// TIA Portal V15.1 export
// export: Created 2024-06-21T08:41:00.3129573Z, ExportSetting WithDefaults, DisplayName Totally Integrated Automation Portal, DisplayVersion V15.1 Update 5, DisplayName TIA Portal Openness, DisplayVersion V15.1 Update 5, DisplayName SINAMICS Startdrive Advanced, DisplayVersion V15.1, DisplayName G130, G150, S120, S150, SINAMICS MV, S210, DisplayVersion V15.1, DisplayName G110M, G120, G120C, G120D, G120P, DisplayVersion V15.1, DisplayName STEP 7 Professional, DisplayVersion V15.1 Update 5, DisplayName STEP 7 Safety, DisplayVersion V15.1, DisplayName WinCC Professional, DisplayVersion V15.1 Update 5, DisplayName SIMATIC Visualization Architect, DisplayVersion V15.1
FUNCTION_BLOCK "LVDComMasterS7-1500"   // FB2210, FBD
TITLE = LVDComMasterPNS7-1500
{ S7_Optimized_Access := 'FALSE' }
AUTHOR : VCC
FAMILY : Communic
VERSION : 0.1
// =============================================================================
// This module Is Used To Read & Send Data With VDCom Protocol
// =============================================================================
// stored: AutoNumber false, IsIECCheckEnabled false, SetENOAutomatically False, UDAEnableTagReadback false
   VAR_INPUT
      I_VDCommRecvDB { ExternalAccessible := 'False'; ExternalVisible := 'False'; ExternalWritable := 'False'} : DB_ANY;   // VD Communication Master DB
      I_VDCommSendDB { ExternalAccessible := 'False'; ExternalVisible := 'False'; ExternalWritable := 'False'} : DB_ANY;   // VD Communication Master DB
   END_VAR
   VAR_OUTPUT
      O_AlarmA { ExternalAccessible := 'False'; ExternalVisible := 'False'; ExternalWritable := 'False'} : Bool;   // Alarm A
      O_AlarmB { ExternalAccessible := 'False'; ExternalVisible := 'False'; ExternalWritable := 'False'} : Bool;   // Alarm B
      O_AlarmC { ExternalAccessible := 'False'; ExternalVisible := 'False'; ExternalWritable := 'False'} : Bool;   // Alarm C
      O_AlarmD { ExternalAccessible := 'False'; ExternalVisible := 'False'; ExternalWritable := 'False'} : Bool;   // Alarm D
      H_AlarmWord { ExternalAccessible := 'False'; ExternalVisible := 'False'; ExternalWritable := 'False'} : DWord;   // HMI Animation
   END_VAR
   VAR_IN_OUT
      IO_Alarm : "Alarm";   // Alarm
      IO_VD : "VDComm";
      IO_ConnectionSetting : Variant;   // Software Connection Settings
      "H_VDComMasterPNS7-1500" : "H_VDComMasterPNS7-1500";   // Animation
   END_VAR
   VAR DB_SPECIFIC
      AD_SendTimeOut { ExternalAccessible := 'False'; ExternalVisible := 'False'; ExternalWritable := 'False'} : Bool;   // Communication Error Send Condition Active Too Long / Kommunikationsfel Sändvillkor Aktivt För Länge
      AD_VersionError { ExternalAccessible := 'False'; ExternalVisible := 'False'; ExternalWritable := 'False'} : Bool;   // Wrong Version Number / Fel Versionsnummer
      AD_ConnError { ExternalAccessible := 'False'; ExternalVisible := 'False'; ExternalWritable := 'False'} : Bool;   // Communication Error Connecting Or Disconnecting / Kommunikationsfel Uppkoppling Eller Nerkoppling
      AD_TCONConnected { ExternalAccessible := 'False'; ExternalVisible := 'False'; ExternalWritable := 'False'} : Bool;   // Not Connected / Ej Uppkopplad
      AD_TSENDError { ExternalAccessible := 'False'; ExternalVisible := 'False'; ExternalWritable := 'False'} : Bool;   // Error Transmission / Fel Sändning
      AD_TRECVError { ExternalAccessible := 'False'; ExternalVisible := 'False'; ExternalWritable := 'False'} : Bool;   // Error Receiving / Fel Mottagning
      AD_NoAckReceived { ExternalAccessible := 'False'; ExternalVisible := 'False'; ExternalWritable := 'False'} : Bool;   // Error On Ack Message / Fel Vid Ack Meddelande
      AD_SequenceNumberNok { ExternalAccessible := 'False'; ExternalVisible := 'False'; ExternalWritable := 'False'} : Bool;   // Incorrect Sequence Number / Felaktigt Sekvensnummer
      AD_TimeoutApplMsgMem { ExternalAccessible := 'False'; ExternalVisible := 'False'; ExternalWritable := 'False'} : Bool;   // Timeout Message To Subsystem / Timeout Meddelande Till Subsystem
      HMIManual { ExternalAccessible := 'False'; ExternalVisible := 'False'; ExternalWritable := 'False'} : Bool;   // Connect or disconnect manual via HMI
      HMIResetAndInit { ExternalAccessible := 'False'; ExternalVisible := 'False'; ExternalWritable := 'False'} : Bool;   // Reset Alarms from HMI
      HMIConnect { ExternalAccessible := 'False'; ExternalVisible := 'False'; ExternalWritable := 'False'} : Bool;   // Connect from HMI
      HMIDisConnect { ExternalAccessible := 'False'; ExternalVisible := 'False'; ExternalWritable := 'False'} : Bool;   // DisConnect from HMI
      Manual { ExternalAccessible := 'False'; ExternalVisible := 'False'; ExternalWritable := 'False'} : Bool;   // Connect or disconnect manual via HMI
      SendActive { ExternalAccessible := 'False'; ExternalVisible := 'False'; ExternalWritable := 'False'} : Bool;   // Sending is Active
      NdrDelayed { ExternalAccessible := 'False'; ExternalVisible := 'False'; ExternalWritable := 'False'} : Bool;   // Time required to elapse before to send acknowledge
      KeepAliveReq { ExternalAccessible := 'False'; ExternalVisible := 'False'; ExternalWritable := 'False'} : Bool;   // Request to send keep alive message
      AckRcvd { ExternalAccessible := 'False'; ExternalVisible := 'False'; ExternalWritable := 'False'} : Bool;   // Acknowledge Received
      SeqNbrOk { ExternalAccessible := 'False'; ExternalVisible := 'False'; ExternalWritable := 'False'} : Bool;   // Sequence number in received message is the same as sended
      AckOk { ExternalAccessible := 'False'; ExternalVisible := 'False'; ExternalWritable := 'False'} : Bool;   // Received acknowledge message ok
      AckNok { ExternalAccessible := 'False'; ExternalVisible := 'False'; ExternalWritable := 'False'} : Bool;   // Received acknowledge message not ok
      NewMessage { ExternalAccessible := 'False'; ExternalVisible := 'False'; ExternalWritable := 'False'} : Bool;   // New Data Message has been received
      SendInactive { ExternalAccessible := 'False'; ExternalVisible := 'False'; ExternalWritable := 'False'} : Bool;   // Sending inActive
      SendJobCompleted { ExternalAccessible := 'False'; ExternalVisible := 'False'; ExternalWritable := 'False'} : Bool;   // Status of the TSEND module: Job Completed no job active
      SendStartOfProc { ExternalAccessible := 'False'; ExternalVisible := 'False'; ExternalWritable := 'False'} : Bool;   // Status of TSEND: Start of Processing
      SendFollowOnCall { ExternalAccessible := 'False'; ExternalVisible := 'False'; ExternalWritable := 'False'} : Bool;   // Status of TSEND: Followon calls being processed
      SendNackMem { ExternalAccessible := 'False'; ExternalVisible := 'False'; ExternalWritable := 'False'} : Bool;   // Command to send Not acknowledge message
      SendNackPulse { ExternalAccessible := 'False'; ExternalVisible := 'False'; ExternalWritable := 'False'} : Bool;   // Pulse to send the Not Acknowledge message
      SendNackCmd { ExternalAccessible := 'False'; ExternalVisible := 'False'; ExternalWritable := 'False'} : Bool;   // Command to send a NOT Acknowledge message
      SendAckMem { ExternalAccessible := 'False'; ExternalVisible := 'False'; ExternalWritable := 'False'} : Bool;   // Command to send Acknowledge message
      SendAckPulse { ExternalAccessible := 'False'; ExternalVisible := 'False'; ExternalWritable := 'False'} : Bool;   // Pulse to send Acknowledge message
      SendAckCmd { ExternalAccessible := 'False'; ExternalVisible := 'False'; ExternalWritable := 'False'} : Bool;   // Command to send an Acknowledge message
      SendKeepAliveMem { ExternalAccessible := 'False'; ExternalVisible := 'False'; ExternalWritable := 'False'} : Bool;   // Command to send the keep alive signal
      SendKeepAlivePulse { ExternalAccessible := 'False'; ExternalVisible := 'False'; ExternalWritable := 'False'} : Bool;   // Pulse to send keep alive message
      SendKeepAliveCmd { ExternalAccessible := 'False'; ExternalVisible := 'False'; ExternalWritable := 'False'} : Bool;   // Command to Send Keep Alive message
      SendApplMsgMem { ExternalAccessible := 'False'; ExternalVisible := 'False'; ExternalWritable := 'False'} : Bool;   // Command to send apllication data
      SendApplMsgPulse { ExternalAccessible := 'False'; ExternalVisible := 'False'; ExternalWritable := 'False'} : Bool;   // Pulse created upon SendApplMsgCmd
      SendApplMsgCmd { ExternalAccessible := 'False'; ExternalVisible := 'False'; ExternalWritable := 'False'} : Bool;   // Command to send an Application message
      NewMsgNbr { ExternalAccessible := 'False'; ExternalVisible := 'False'; ExternalWritable := 'False'} : Bool;   // Message number of last received message
      NackIsLastSent { ExternalAccessible := 'False'; ExternalVisible := 'False'; ExternalWritable := 'False'} : Bool;   // Memorise that Nack was send
      DupplMsg { ExternalAccessible := 'False'; ExternalVisible := 'False'; ExternalWritable := 'False'} : Bool;   // When received msg number is the same as previous
      RecvLenOK { ExternalAccessible := 'False'; ExternalVisible := 'False'; ExternalWritable := 'False'} : Bool;   // If protocol Len and actual received msg are the same
      WaitForAck { ExternalAccessible := 'False'; ExternalVisible := 'False'; ExternalWritable := 'False'} : Bool;   // State waiting for acknowledge
      TimeOutTConn { ExternalAccessible := 'False'; ExternalVisible := 'False'; ExternalWritable := 'False'} : Bool;   // Time out on connecting or disconnecting
      TimeoutTCON { ExternalAccessible := 'False'; ExternalVisible := 'False'; ExternalWritable := 'False'} : Bool;   // Memory of connection time out
      TimeoutTDISCON { ExternalAccessible := 'False'; ExternalVisible := 'False'; ExternalWritable := 'False'} : Bool;   // Time out on disconnecting
      TimeoutApplMsg { ExternalAccessible := 'False'; ExternalVisible := 'False'; ExternalWritable := 'False'} : Bool;   // Time Out on apllication message, no ack received
      DisconnConn { ExternalAccessible := 'False'; ExternalVisible := 'False'; ExternalWritable := 'False'} : Bool;   // Time before connecting after disconnecting
      Edge { ExternalAccessible := 'False'; ExternalVisible := 'False'; ExternalWritable := 'False'} : Bool;   // Positive edge Detection for connected
      ResetAppliMsgCnt { ExternalAccessible := 'False'; ExternalVisible := 'False'; ExternalWritable := 'False'} : Bool;   // Reset the Application message counter
      ResetKeepAliveCnt { ExternalAccessible := 'False'; ExternalVisible := 'False'; ExternalWritable := 'False'} : Bool;   // Reset the keep alive counter
      ResetAckCmdCnt { ExternalAccessible := 'False'; ExternalVisible := 'False'; ExternalWritable := 'False'} : Bool;   // Reset the acknowledge counter
      ResetNackCmdCnt { ExternalAccessible := 'False'; ExternalVisible := 'False'; ExternalWritable := 'False'} : Bool;   // Reset the Nacknowledge counter
      ResetAckRcvCnt { ExternalAccessible := 'False'; ExternalVisible := 'False'; ExternalWritable := 'False'} : Bool;   // Reset the received Ack counter
      ResetDataMsgCnt { ExternalAccessible := 'False'; ExternalVisible := 'False'; ExternalWritable := 'False'} : Bool;   // Reset the received Data message counter
      ResetSeqNokCnt { ExternalAccessible := 'False'; ExternalVisible := 'False'; ExternalWritable := 'False'} : Bool;   // Reset the sequence nok counter
      ResetSendActive { ExternalAccessible := 'False'; ExternalVisible := 'False'; ExternalWritable := 'False'} : Bool;   // Reset Send Active due to time out
      SendDone { ExternalAccessible := 'False'; ExternalVisible := 'False'; ExternalWritable := 'False'} : Bool;   // Reset the Ndr counter on overrun
      DelayOpen { ExternalAccessible := 'False'; ExternalVisible := 'False'; ExternalWritable := 'False'} : Bool;   // Delay Start Connect
      DelayConn { ExternalAccessible := 'False'; ExternalVisible := 'False'; ExternalWritable := 'False'} : Bool;   // Delay Connected
      AlarmA { ExternalAccessible := 'False'; ExternalVisible := 'False'; ExternalWritable := 'False'} : Bool;   // Alarm A
      AlarmB { ExternalAccessible := 'False'; ExternalVisible := 'False'; ExternalWritable := 'False'} : Bool;   // Alarm B
      AlarmC { ExternalAccessible := 'False'; ExternalVisible := 'False'; ExternalWritable := 'False'} : Bool;   // Alarm C
      AlarmD { ExternalAccessible := 'False'; ExternalVisible := 'False'; ExternalWritable := 'False'} : Bool;   // Alarm D
      OldSubSystem { ExternalAccessible := 'False'; ExternalVisible := 'False'; ExternalWritable := 'False'} : Word;   // Memorise last received subsystem address
      OldRecMsgNbr { ExternalAccessible := 'False'; ExternalVisible := 'False'; ExternalWritable := 'False'} : Word := W#16#999;   // Memorise the last message number
      SendMsgNbr { ExternalAccessible := 'False'; ExternalVisible := 'False'; ExternalWritable := 'False'} : Word;   // Number is incremented for each msg and Reset to 1 when > 1000
      RecvLen { ExternalAccessible := 'False'; ExternalVisible := 'False'; ExternalWritable := 'False'} : Int;   // Memory of the received data length
      RecvDBNbr { ExternalAccessible := 'False'; ExternalVisible := 'False'; ExternalWritable := 'False'} : Int;   // Receive DB Number
      SendDBNbr { ExternalAccessible := 'False'; ExternalVisible := 'False'; ExternalWritable := 'False'} : Int;   // Send DB Number
      SendApplMsgCnt { ExternalAccessible := 'False'; ExternalVisible := 'False'; ExternalWritable := 'False'} : Int;   // Counting number of Application messages
      SendKeepAliveCnt { ExternalAccessible := 'False'; ExternalVisible := 'False'; ExternalWritable := 'False'} : Int;   // Counting number of keep alive messages
      SendAckCmdCnt { ExternalAccessible := 'False'; ExternalVisible := 'False'; ExternalWritable := 'False'} : Int;   // Counting the number of Ack messages
      SendNackCmdCnt { ExternalAccessible := 'False'; ExternalVisible := 'False'; ExternalWritable := 'False'} : Int;   // Counting the number of Nack messages
      RcvAckCnt { ExternalAccessible := 'False'; ExternalVisible := 'False'; ExternalWritable := 'False'} : Int;   // Counting the number of received Ack messages
      RcvDataMsgCnt { ExternalAccessible := 'False'; ExternalVisible := 'False'; ExternalWritable := 'False'} : Int;   // Counting the number of Data messages
      SeqNokCnt { ExternalAccessible := 'False'; ExternalVisible := 'False'; ExternalWritable := 'False'} : Int;   // Counter indicating the number of received sequence errors
      NdrCnt { ExternalAccessible := 'False'; ExternalVisible := 'False'; ExternalWritable := 'False'} : Int;   // Counter indicating the all received events
   END_VAR
   VAR
      TConVD { ExternalAccessible := 'False'; ExternalVisible := 'False'; ExternalWritable := 'False'; S7_SetPoint := 'True'} : TCON;   // Connect
      TDisConVD { ExternalAccessible := 'False'; ExternalVisible := 'False'; ExternalWritable := 'False'; S7_SetPoint := 'True'} : TDISCON;   // Disconnect
      TRcvVDData { ExternalAccessible := 'False'; ExternalVisible := 'False'; ExternalWritable := 'False'; S7_SetPoint := 'True'} : TRCV;   // Receive
      TSendVD { ExternalAccessible := 'False'; ExternalVisible := 'False'; ExternalWritable := 'False'; S7_SetPoint := 'True'} : TSEND;   // Send
   END_VAR
   VAR DB_SPECIFIC
      TCON { ExternalAccessible := 'False'; ExternalVisible := 'False'; ExternalWritable := 'False'} : Struct   // Structure
         Connecting { ExternalAccessible := 'False'; ExternalVisible := 'False'; ExternalWritable := 'False'} : Bool;
         Connected { ExternalAccessible := 'False'; ExternalVisible := 'False'; ExternalWritable := 'False'} : Bool;
         Done { ExternalAccessible := 'False'; ExternalVisible := 'False'; ExternalWritable := 'False'} : Bool;
         Busy { ExternalAccessible := 'False'; ExternalVisible := 'False'; ExternalWritable := 'False'} : Bool;
         Error { ExternalAccessible := 'False'; ExternalVisible := 'False'; ExternalWritable := 'False'} : Bool;
         Req { ExternalAccessible := 'False'; ExternalVisible := 'False'; ExternalWritable := 'False'} : Bool;
         Status { ExternalAccessible := 'False'; ExternalVisible := 'False'; ExternalWritable := 'False'} : Word;
         Status_Mem { ExternalAccessible := 'False'; ExternalVisible := 'False'; ExternalWritable := 'False'} : Word;
         Status_Int { ExternalAccessible := 'False'; ExternalVisible := 'False'; ExternalWritable := 'False'} : Int;
      END_STRUCT;
      TDISCON { ExternalAccessible := 'False'; ExternalVisible := 'False'; ExternalWritable := 'False'} : Struct   // Structure
         Disconnecting { ExternalAccessible := 'False'; ExternalVisible := 'False'; ExternalWritable := 'False'} : Bool;
         Done { ExternalAccessible := 'False'; ExternalVisible := 'False'; ExternalWritable := 'False'} : Bool;
         Busy { ExternalAccessible := 'False'; ExternalVisible := 'False'; ExternalWritable := 'False'} : Bool;
         Error { ExternalAccessible := 'False'; ExternalVisible := 'False'; ExternalWritable := 'False'} : Bool;
         Req { ExternalAccessible := 'False'; ExternalVisible := 'False'; ExternalWritable := 'False'} : Bool;
         Status { ExternalAccessible := 'False'; ExternalVisible := 'False'; ExternalWritable := 'False'} : Word;
         Status_Mem { ExternalAccessible := 'False'; ExternalVisible := 'False'; ExternalWritable := 'False'} : Word;
      END_STRUCT;
      TRECV { ExternalAccessible := 'False'; ExternalVisible := 'False'; ExternalWritable := 'False'} : Struct   // Structure
         Receiving { ExternalAccessible := 'False'; ExternalVisible := 'False'; ExternalWritable := 'False'} : Bool;
         Ndr { ExternalAccessible := 'False'; ExternalVisible := 'False'; ExternalWritable := 'False'} : Bool;
         Busy { ExternalAccessible := 'False'; ExternalVisible := 'False'; ExternalWritable := 'False'} : Bool;
         Error { ExternalAccessible := 'False'; ExternalVisible := 'False'; ExternalWritable := 'False'} : Bool;
         RcvConError { ExternalAccessible := 'False'; ExternalVisible := 'False'; ExternalWritable := 'False'} : Bool;
         Status { ExternalAccessible := 'False'; ExternalVisible := 'False'; ExternalWritable := 'False'} : Word;
         Status_Mem { ExternalAccessible := 'False'; ExternalVisible := 'False'; ExternalWritable := 'False'} : Word;
         Length { ExternalAccessible := 'False'; ExternalVisible := 'False'; ExternalWritable := 'False'} : UDInt;
      END_STRUCT;
      TSEND { ExternalAccessible := 'False'; ExternalVisible := 'False'; ExternalWritable := 'False'} : Struct   // Structure
         Sending { ExternalAccessible := 'False'; ExternalVisible := 'False'; ExternalWritable := 'False'} : Bool;
         Done { ExternalAccessible := 'False'; ExternalVisible := 'False'; ExternalWritable := 'False'} : Bool;
         Busy { ExternalAccessible := 'False'; ExternalVisible := 'False'; ExternalWritable := 'False'} : Bool;
         Error { ExternalAccessible := 'False'; ExternalVisible := 'False'; ExternalWritable := 'False'} : Bool;
         Status { ExternalAccessible := 'False'; ExternalVisible := 'False'; ExternalWritable := 'False'} : Word;
         Status_Mem { ExternalAccessible := 'False'; ExternalVisible := 'False'; ExternalWritable := 'False'} : Word;
      END_STRUCT;
      NackCmdCntr { ExternalAccessible := 'False'; ExternalVisible := 'False'; ExternalWritable := 'False'; S7_SetPoint := 'True'} : CTU_INT;   // Count number of NotAck messages send by PLC
      AckCmdCnt { ExternalAccessible := 'False'; ExternalVisible := 'False'; ExternalWritable := 'False'; S7_SetPoint := 'True'} : CTU_INT;   // Count number of Ack messages send by PLC
      KeepAliveCnt { ExternalAccessible := 'False'; ExternalVisible := 'False'; ExternalWritable := 'False'; S7_SetPoint := 'True'} : CTU_INT;   // Count number of Keep Alived Messages send by PLC
      AppliMsgCnt { ExternalAccessible := 'False'; ExternalVisible := 'False'; ExternalWritable := 'False'; S7_SetPoint := 'True'} : CTU_INT;   // Count number of Application messages send by PLC
      AckRvcCntr { ExternalAccessible := 'False'; ExternalVisible := 'False'; ExternalWritable := 'False'; S7_SetPoint := 'True'} : CTU_INT;   // Count number of Ack messages received
      DataMsgRcvCntr { ExternalAccessible := 'False'; ExternalVisible := 'False'; ExternalWritable := 'False'; S7_SetPoint := 'True'} : CTU_INT;   // Count number of data messages received
      SeqNumNok { ExternalAccessible := 'False'; ExternalVisible := 'False'; ExternalWritable := 'False'; S7_SetPoint := 'True'} : CTU_INT;   // counter to know the sequence number errors
      NdrPace { ExternalAccessible := 'False'; ExternalVisible := 'False'; ExternalWritable := 'False'; S7_SetPoint := 'True'} : TOF_TIME;   // Make sure that not too many messages are received at once
      TimeOutSending { ExternalAccessible := 'False'; ExternalVisible := 'False'; ExternalWritable := 'False'; S7_SetPoint := 'True'} : TON_TIME;   // TimeOut on Send operation
      TimeOutAckApplMsg { ExternalAccessible := 'False'; ExternalVisible := 'False'; ExternalWritable := 'False'; S7_SetPoint := 'True'} : TON_TIME;   // Timeout on reception of Ack on Application message
      TimeOutOnConnection { ExternalAccessible := 'False'; ExternalVisible := 'False'; ExternalWritable := 'False'; S7_SetPoint := 'True'} : TON_TIME;   // TimeOut on connecting
      KeepAliveFreq { ExternalAccessible := 'False'; ExternalVisible := 'False'; ExternalWritable := 'False'; S7_SetPoint := 'True'} : TON_TIME;   // Timer to timeout the keep alive messages
      DisconnectRequest { ExternalAccessible := 'False'; ExternalVisible := 'False'; ExternalWritable := 'False'; S7_SetPoint := 'True'} : TON_TIME;   // Request to disconnect after timeout
      WaitingForAck { ExternalAccessible := 'False'; ExternalVisible := 'False'; ExternalWritable := 'False'; S7_SetPoint := 'True'} : TON_TIME;   // Waiting for Ack to receive
      SubSystResponseTimeOut { ExternalAccessible := 'False'; ExternalVisible := 'False'; ExternalWritable := 'False'; S7_SetPoint := 'True'} : TON_TIME;   // TimeOut subsystem reply
      TimeOutSendActive { ExternalAccessible := 'False'; ExternalVisible := 'False'; ExternalWritable := 'False'; S7_SetPoint := 'True'} : TON_TIME;   // When SendActive is ON for too long
      DelayStartConnect { ExternalAccessible := 'False'; ExternalVisible := 'False'; ExternalWritable := 'False'; S7_SetPoint := 'True'} : TON_TIME;   // FB
      DelayConnected { ExternalAccessible := 'False'; ExternalVisible := 'False'; ExternalWritable := 'False'; S7_SetPoint := 'True'} : TON_TIME;   // FB
   END_VAR
   VAR
      _VDConManual { ExternalAccessible := 'False'; ExternalVisible := 'False'; ExternalWritable := 'False'; S7_SetPoint := 'True'} : "LToggle";   // FB
   END_VAR
   VAR DB_SPECIFIC
      ConnectionSettings { ExternalAccessible := 'False'; ExternalVisible := 'False'; ExternalWritable := 'False'; S7_SetPoint := 'True'} : TCON_Param;   // Structrure
   END_VAR
   VAR_TEMP
      PointerRecv : Any;   // Pointer to receive buffer
      PointerSend : Any;   // Pointer to Send Buffer
      PointerSendBuf : Any;   // Pointer to Send buffer
      OutBuf : Int;   // Integer to select the Send buffer
      UserMsgType : Bool;   // Message Type
      RecvTimeOut : Bool;   // Receive Time Out
      MsgLen : UDInt;   // Message length
      MessageLengthRecv : Int;   // Message Length receive
      TempIntStatus : Int;   // for type casting to integer
      TempInt : Int;   // for type casting to integer
      RecvDBNO : UInt;
      LengthDB : UDInt;
      TempBool : Array[1..16] of Bool;
      ConnectionSetting : Variant;
   END_VAR
   VAR_TEMP   // added for the SCL form of the ladder/FBD networks
      _w1 : Bool;
      _w2 : Bool;
   END_VAR
BEGIN

REGION Network 1: **** 1 - Inputs **** Extract the selection from HMI
   // Extract the selection from HMI
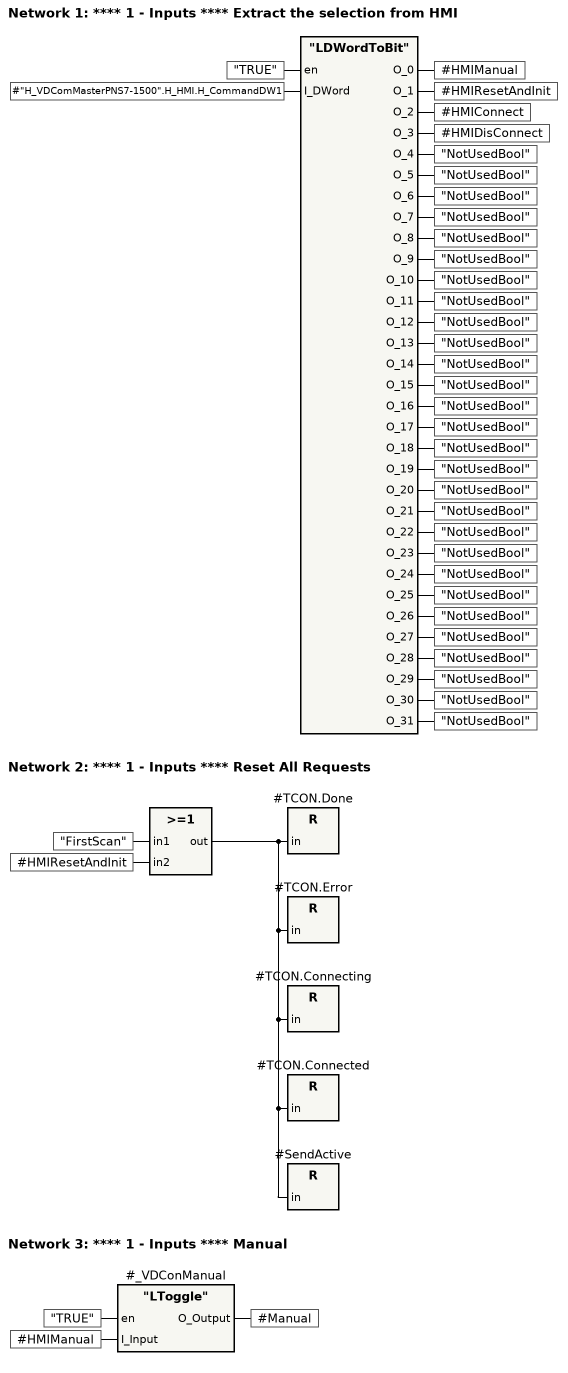
   IF "TRUE" THEN
       "LDWordToBit"(I_DWord := #"H_VDComMasterPNS7-1500".H_HMI.H_CommandDW1,
                     O_0 => #HMIManual,
                     O_1 => #HMIResetAndInit,
                     O_2 => #HMIConnect,
                     O_3 => #HMIDisConnect,
                     O_4 => "NotUsedBool",
                     O_5 => "NotUsedBool",
                     O_6 => "NotUsedBool",
                     O_7 => "NotUsedBool",
                     O_8 => "NotUsedBool",
                     O_9 => "NotUsedBool",
                     O_10 => "NotUsedBool",
                     O_11 => "NotUsedBool",
                     O_12 => "NotUsedBool",
                     O_13 => "NotUsedBool",
                     O_14 => "NotUsedBool",
                     O_15 => "NotUsedBool",
                     O_16 => "NotUsedBool",
                     O_17 => "NotUsedBool",
                     O_18 => "NotUsedBool",
                     O_19 => "NotUsedBool",
                     O_20 => "NotUsedBool",
                     O_21 => "NotUsedBool",
                     O_22 => "NotUsedBool",
                     O_23 => "NotUsedBool",
                     O_24 => "NotUsedBool",
                     O_25 => "NotUsedBool",
                     O_26 => "NotUsedBool",
                     O_27 => "NotUsedBool",
                     O_28 => "NotUsedBool",
                     O_29 => "NotUsedBool",
                     O_30 => "NotUsedBool",
                     O_31 => "NotUsedBool");
   END_IF;
END_REGION

REGION Network 2: **** 1 - Inputs **** Reset All Requests
   // Reset All Requests
   IF "FirstScan" OR #HMIResetAndInit THEN
       #TCON.Done := FALSE;
       #TCON.Error := FALSE;
       #TCON.Connecting := FALSE;
       #TCON.Connected := FALSE;
       #SendActive := FALSE;
   END_IF;
END_REGION

REGION Network 3: **** 1 - Inputs **** Manual
   // Manual
   IF "TRUE" THEN
       #_VDConManual(I_Input := #HMIManual, O_Output => #Manual);   // "LToggle"
   END_IF;
END_REGION

REGION Network 4: **** 1 - Inputs **** Reset Com Disconnect
   // Reset Com Disconnect
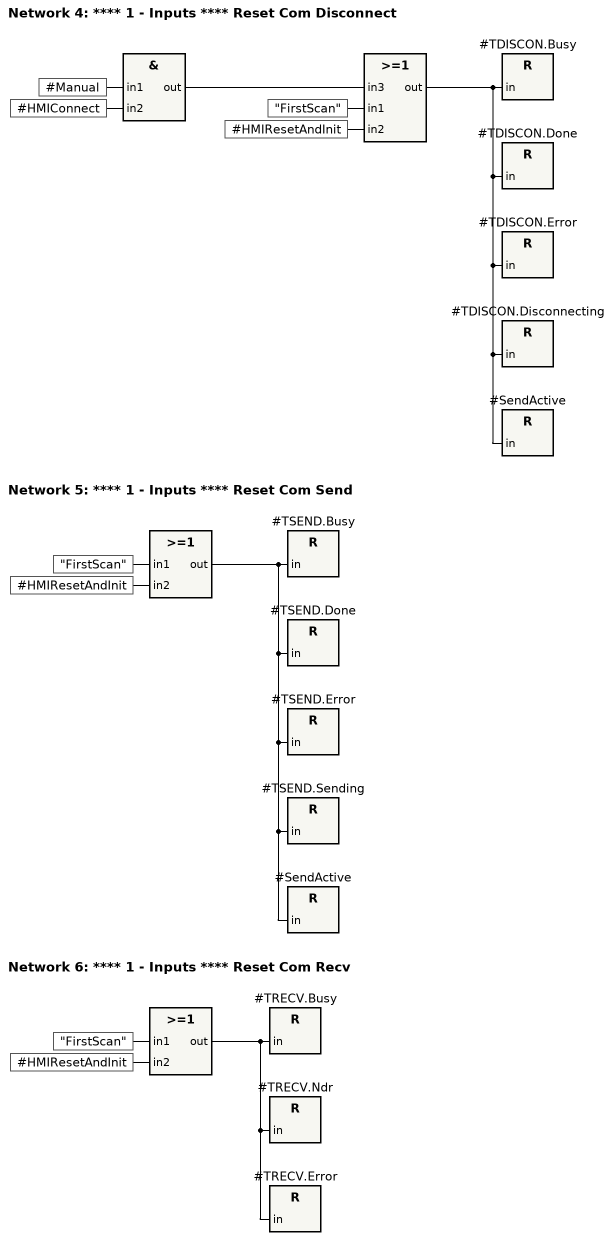
   IF (#Manual AND #HMIConnect) OR "FirstScan" OR #HMIResetAndInit THEN
       #TDISCON.Busy := FALSE;
       #TDISCON.Done := FALSE;
       #TDISCON.Error := FALSE;
       #TDISCON.Disconnecting := FALSE;
       #SendActive := FALSE;
   END_IF;
END_REGION

REGION Network 5: **** 1 - Inputs **** Reset Com Send
   // Reset com Send
   IF "FirstScan" OR #HMIResetAndInit THEN
       #TSEND.Busy := FALSE;
       #TSEND.Done := FALSE;
       #TSEND.Error := FALSE;
       #TSEND.Sending := FALSE;
       #SendActive := FALSE;
   END_IF;
END_REGION

REGION Network 6: **** 1 - Inputs **** Reset Com Recv
   // Reset Com Recv
   IF "FirstScan" OR #HMIResetAndInit THEN
       #TRECV.Busy := FALSE;
       #TRECV.Ndr := FALSE;
       #TRECV.Error := FALSE;
   END_IF;
END_REGION

REGION Network 7: **** 3.1 - Communication - Other Systems **** Reset Communications / **** 1 - Inputs **** Reset Communication
   // Reset Communications / Reset communication status words
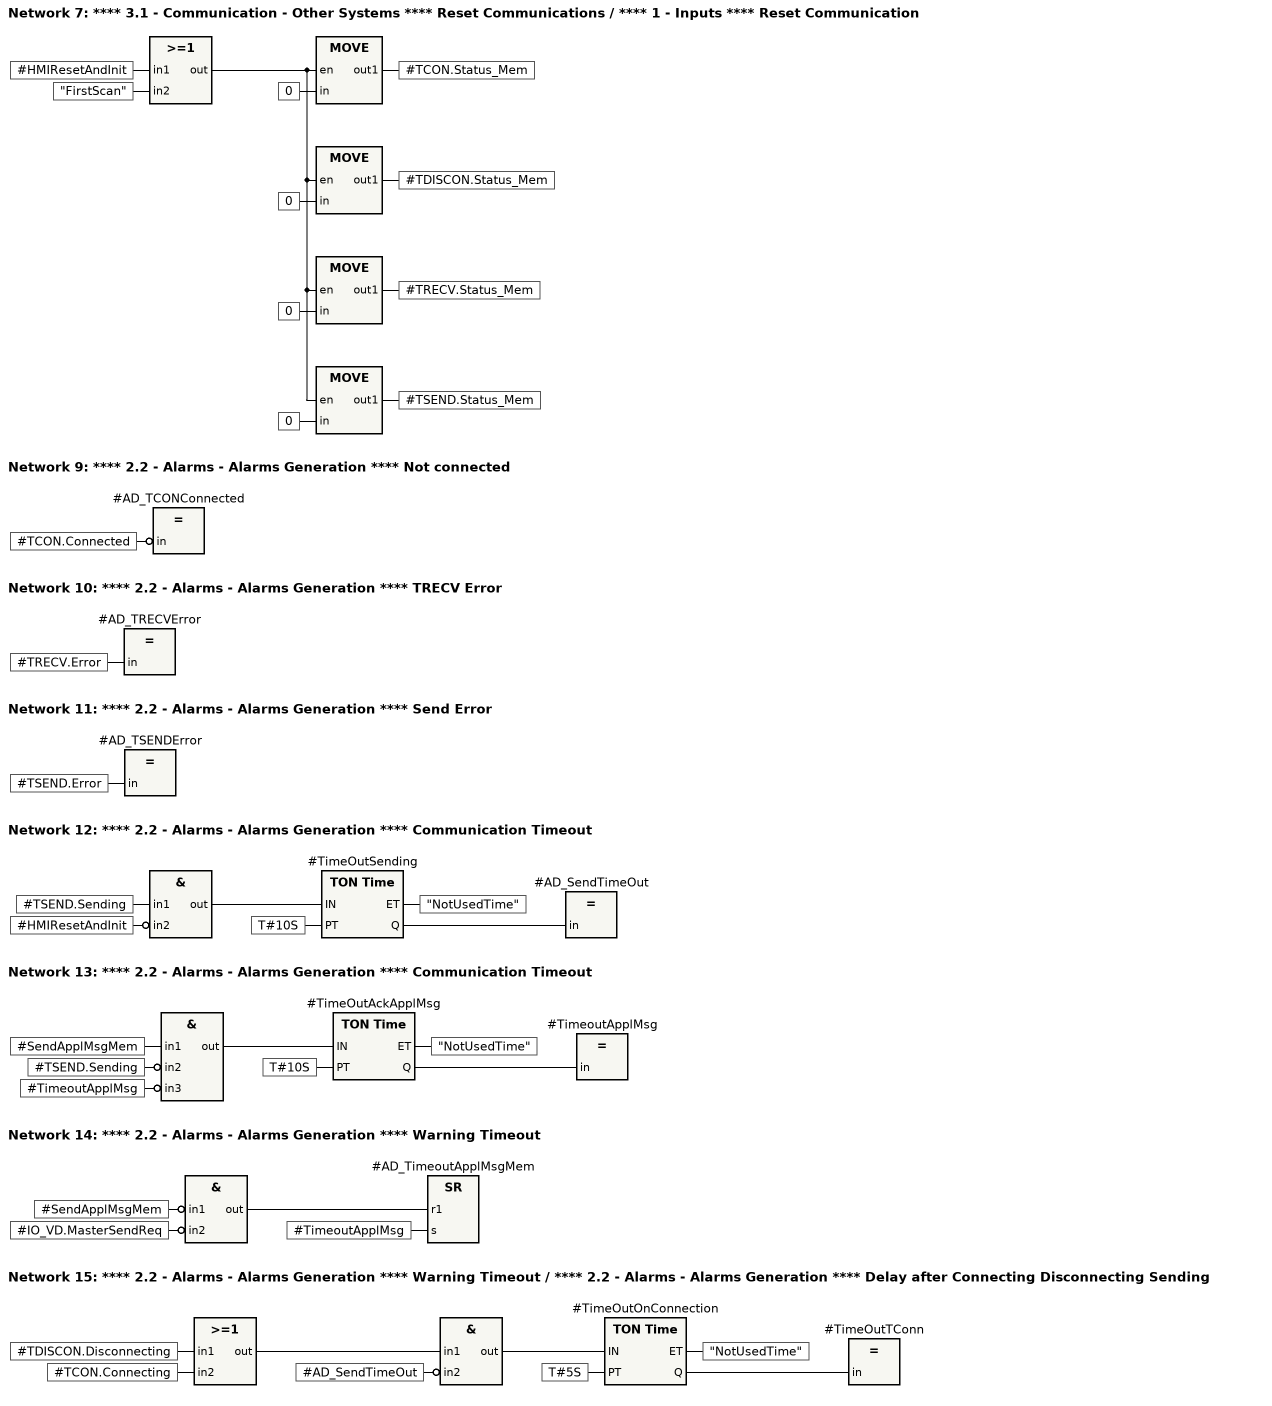
   IF #HMIResetAndInit OR "FirstScan" THEN
       #TCON.Status_Mem := 0;
       #TDISCON.Status_Mem := 0;
       #TRECV.Status_Mem := 0;
       #TSEND.Status_Mem := 0;
   END_IF;
END_REGION

NETWORK
TITLE = **** 1 - Inputs **** Load DB
// Load DB numbers to local variables from the Receive and Send DB
// Read DB Number Receive (VD Master System Receive DB)
      OPN   #I_VDCommRecvDB;
      L     DBNO;
      T     #RecvDBNbr;

// Read DB Number Send (VD Master System Send DB)
      OPN   #I_VDCommSendDB;
      L     DBNO;
      T     #SendDBNbr;



REGION Network 9: **** 2.2 - Alarms - Alarms Generation **** Not connected
   // Not connected
   #AD_TCONConnected := NOT #TCON.Connected;
END_REGION

REGION Network 10: **** 2.2 - Alarms - Alarms Generation **** TRECV Error
   // TRECV Error
   #AD_TRECVError := #TRECV.Error;
END_REGION

REGION Network 11: **** 2.2 - Alarms - Alarms Generation **** Send Error
   // Send Error
   #AD_TSENDError := #TSEND.Error;
END_REGION

REGION Network 12: **** 2.2 - Alarms - Alarms Generation **** Communication Timeout
   // Communication timeout while sending
   #TimeOutSending(IN := #TSEND.Sending AND NOT #HMIResetAndInit, PT := T#10S, ET => "NotUsedTime");   // TON
   #AD_SendTimeOut := #TimeOutSending.Q;
END_REGION

REGION Network 13: **** 2.2 - Alarms - Alarms Generation **** Communication Timeout
   // Communication timeout while Application message
   #TimeOutAckApplMsg(IN := #SendApplMsgMem AND NOT #TSEND.Sending AND NOT #TimeoutApplMsg,   // TON
                      PT := T#10S,
                      ET => "NotUsedTime");
   #TimeoutApplMsg := #TimeOutAckApplMsg.Q;
END_REGION

REGION Network 14: **** 2.2 - Alarms - Alarms Generation **** Warning Timeout
   // Warning Timeout Application message
   IF #TimeoutApplMsg THEN
       #AD_TimeoutApplMsgMem := TRUE;   // SR flip-flop
   END_IF;
   IF NOT #SendApplMsgMem AND NOT #IO_VD.MasterSendReq THEN #AD_TimeoutApplMsgMem := FALSE; END_IF;
END_REGION

REGION Network 15: **** 2.2 - Alarms - Alarms Generation **** Warning Timeout / **** 2.2 - Alarms - Alarms Generation **** Delay after Connecting Disconnecting Sending
   // Warning Timeout Application message / Delay after Connecting Disconnecting Sending
   #TimeOutOnConnection(IN := (#TDISCON.Disconnecting OR #TCON.Connecting) AND NOT #AD_SendTimeOut,   // TON
                        PT := T#5S,
                        ET => "NotUsedTime");
   #TimeOutTConn := #TimeOutOnConnection.Q;
END_REGION

REGION Network 16: **** 2.2 - Alarms - Alarms Generation **** Timeout Keep Alive
   // Timeout Keep Alive
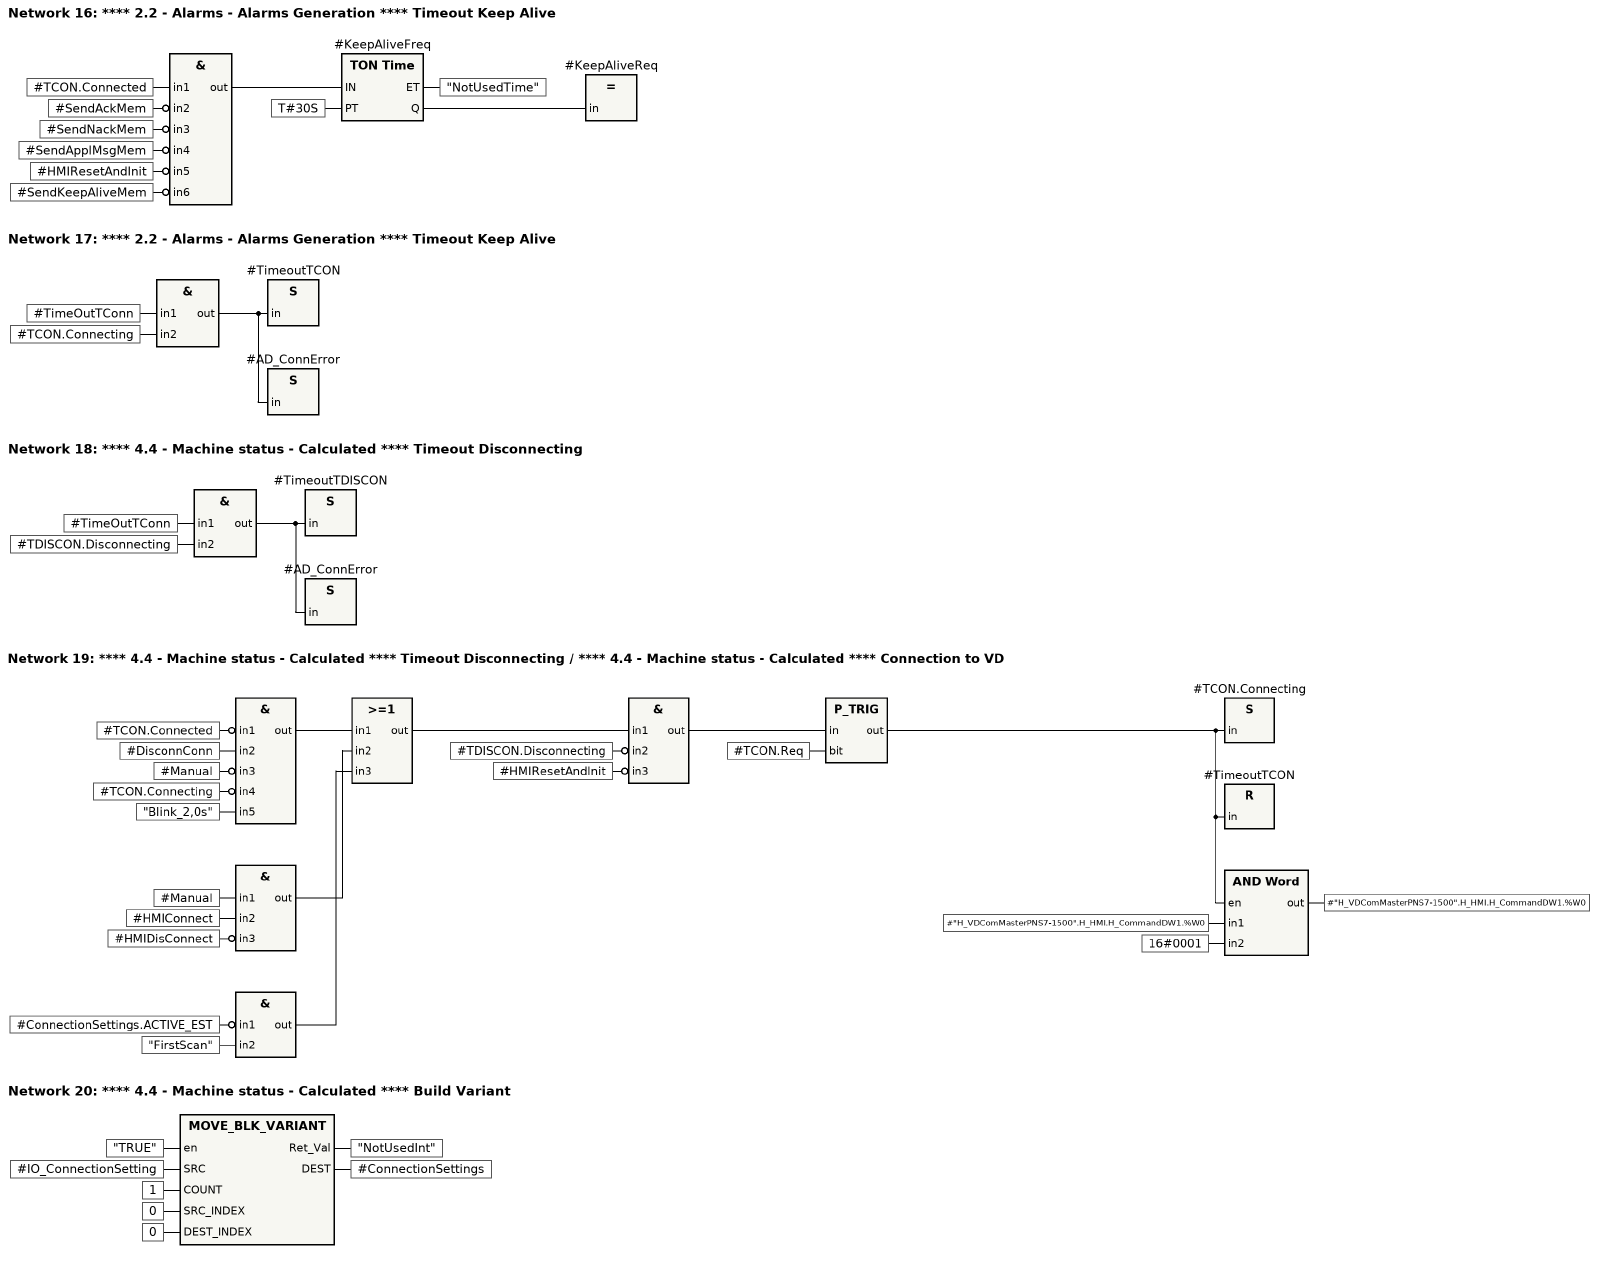
   #KeepAliveFreq(IN := #TCON.Connected AND NOT #SendAckMem AND NOT #SendNackMem AND NOT #SendApplMsgMem AND NOT #HMIResetAndInit AND NOT #SendKeepAliveMem,   // TON
                  PT := T#30S,
                  ET => "NotUsedTime");
   #KeepAliveReq := #KeepAliveFreq.Q;
END_REGION

REGION Network 17: **** 2.2 - Alarms - Alarms Generation **** Timeout Keep Alive
   // Timeout Keep Alive
   IF #TimeOutTConn AND #TCON.Connecting THEN
       #TimeoutTCON := TRUE;
       #AD_ConnError := TRUE;
   END_IF;
END_REGION

REGION Network 18: **** 4.4 - Machine status - Calculated **** Timeout Disconnecting
   // Timeout Disconnecting
   IF #TimeOutTConn AND #TDISCON.Disconnecting THEN
       #TimeoutTDISCON := TRUE;
       #AD_ConnError := TRUE;
   END_IF;
END_REGION

REGION Network 19: **** 4.4 - Machine status - Calculated **** Timeout Disconnecting / **** 4.4 - Machine status - Calculated **** Connection to VD
   // Timeout Disconnecting / Connection to the VD if NOT connecting AND NOT connecte PLC restart and passive connection establishment (to be ready to listen)
   #_w1 := ((NOT #TCON.Connected AND #DisconnConn AND NOT #Manual AND NOT #TCON.Connecting AND "Blink_2,0s") OR (#Manual AND #HMIConnect AND NOT #HMIDisConnect) OR (NOT #ConnectionSettings.ACTIVE_EST AND "FirstScan")) AND NOT #TDISCON.Disconnecting AND NOT #HMIResetAndInit;
   #_w2 := #_w1 AND NOT #TCON.Req;   // rising edge
   #TCON.Req := #_w1;
   IF #_w2 THEN
       #TCON.Connecting := TRUE;
       #TimeoutTCON := FALSE;
       #"H_VDComMasterPNS7-1500".H_HMI.H_CommandDW1.%W0 := #"H_VDComMasterPNS7-1500".H_HMI.H_CommandDW1.%W0 AND 16#0001;
   END_IF;
END_REGION

REGION Network 20: **** 4.4 - Machine status - Calculated **** Build Variant
   // Build Variant
   IF "TRUE" THEN
       "NotUsedInt" := MOVE_BLK_VARIANT(SRC := #IO_ConnectionSetting,
                               COUNT := 1,
                               SRC_INDEX := 0,
                               DEST_INDEX := 0,
                               DEST => #ConnectionSettings);
   END_IF;
END_REGION

REGION Network 21: **** 4.4 - Machine status - Calculated **** Build Variant / **** 4.4 - Machine status - Calculated **** Connection
   // Build Variant / Connection
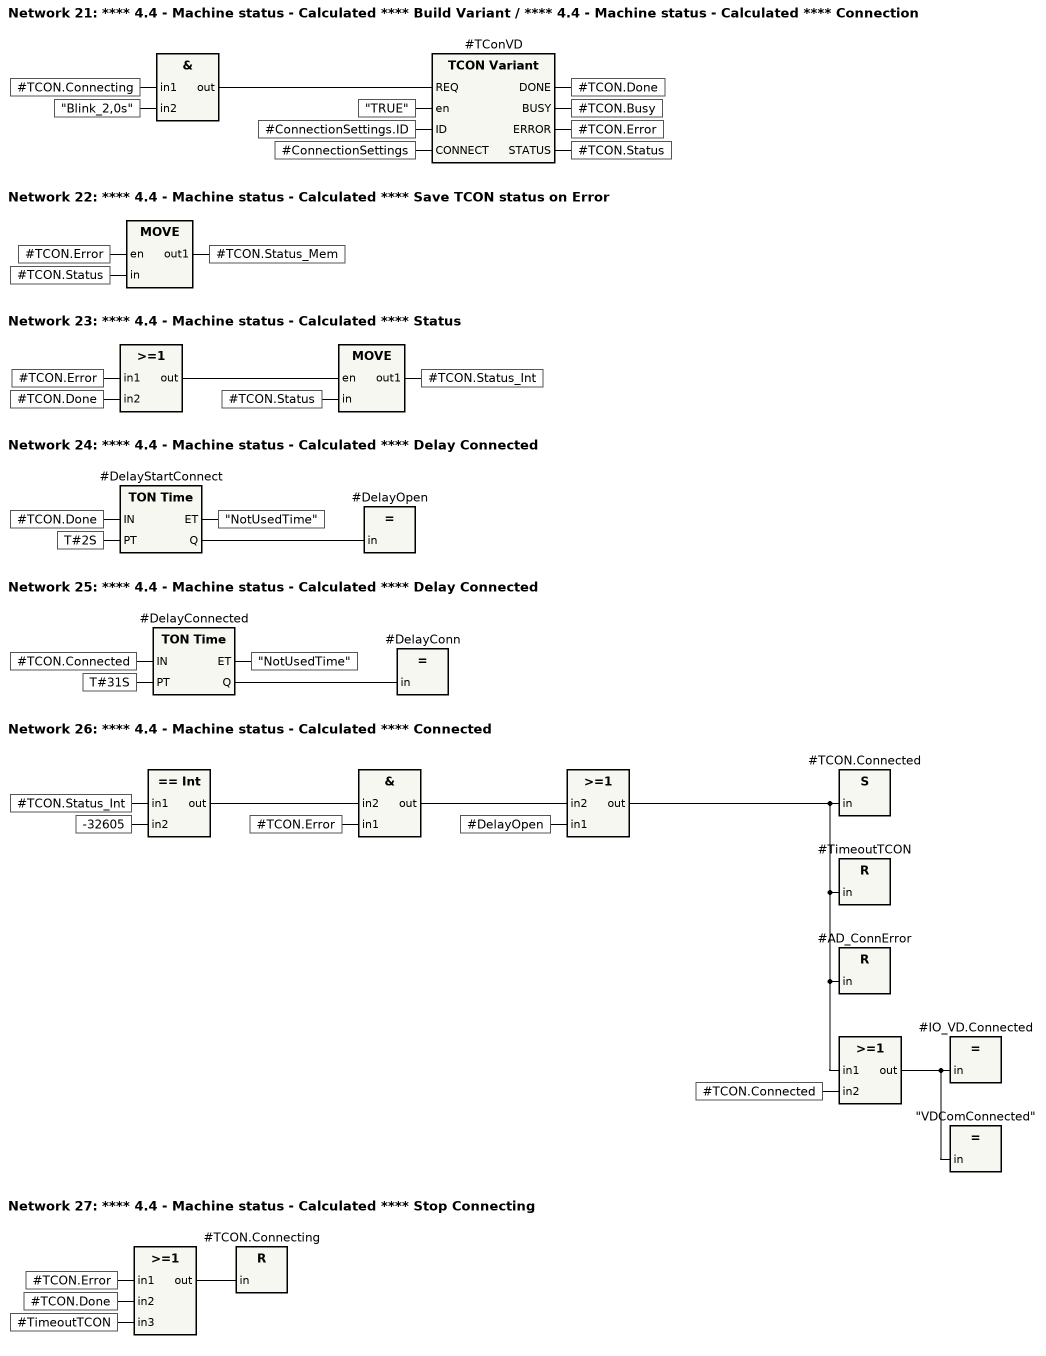
   IF "TRUE" THEN
       #TConVD(REQ := #TCON.Connecting AND "Blink_2,0s",   // TCON
               ID := #ConnectionSettings.ID,
               CONNECT := #ConnectionSettings,
               DONE => #TCON.Done,
               BUSY => #TCON.Busy,
               ERROR => #TCON.Error,
               STATUS => #TCON.Status);
   END_IF;
END_REGION

REGION Network 22: **** 4.4 - Machine status - Calculated **** Save TCON status on Error
   // Save TCON status on Error
   IF #TCON.Error THEN #TCON.Status_Mem := #TCON.Status; END_IF;
END_REGION

REGION Network 23: **** 4.4 - Machine status - Calculated **** Status
   // Status
   IF #TCON.Error OR #TCON.Done THEN #TCON.Status_Int := #TCON.Status; END_IF;
END_REGION

REGION Network 24: **** 4.4 - Machine status - Calculated **** Delay Connected
   // Delay Conected
   #DelayStartConnect(IN := #TCON.Done, PT := T#2S, ET => "NotUsedTime");   // TON
   #DelayOpen := #DelayStartConnect.Q;
END_REGION

REGION Network 25: **** 4.4 - Machine status - Calculated **** Delay Connected
   // Delay Conected
   #DelayConnected(IN := #TCON.Connected, PT := T#31S, ET => "NotUsedTime");   // TON
   #DelayConn := #DelayConnected.Q;
END_REGION

REGION Network 26: **** 4.4 - Machine status - Calculated **** Connected
   // Connected if ,Done bit or if connected already (80A3 = -32605)
   #_w1 := ((#TCON.Status_Int = (-32605)) AND #TCON.Error) OR #DelayOpen;
   IF #_w1 THEN
       #TCON.Connected := TRUE;
       #TimeoutTCON := FALSE;
       #AD_ConnError := FALSE;
   END_IF;
   #IO_VD.Connected := #_w1 OR #TCON.Connected;
   "VDComConnected" := #IO_VD.Connected;
END_REGION

REGION Network 27: **** 4.4 - Machine status - Calculated **** Stop Connecting
   // Stop connecting attempt if Error,Done,Connecting AND NOT Busy
   IF #TCON.Error OR #TCON.Done OR #TimeoutTCON THEN #TCON.Connecting := FALSE; END_IF;
END_REGION

REGION Network 28: **** 4.4 - Machine status - Calculated **** Timeout Disconnecting / **** 4.4 - Machine status - Calculated **** Disconnect on Receive
   // Timeout Disconnecting / Disconnect on Receive error or on HMI Request
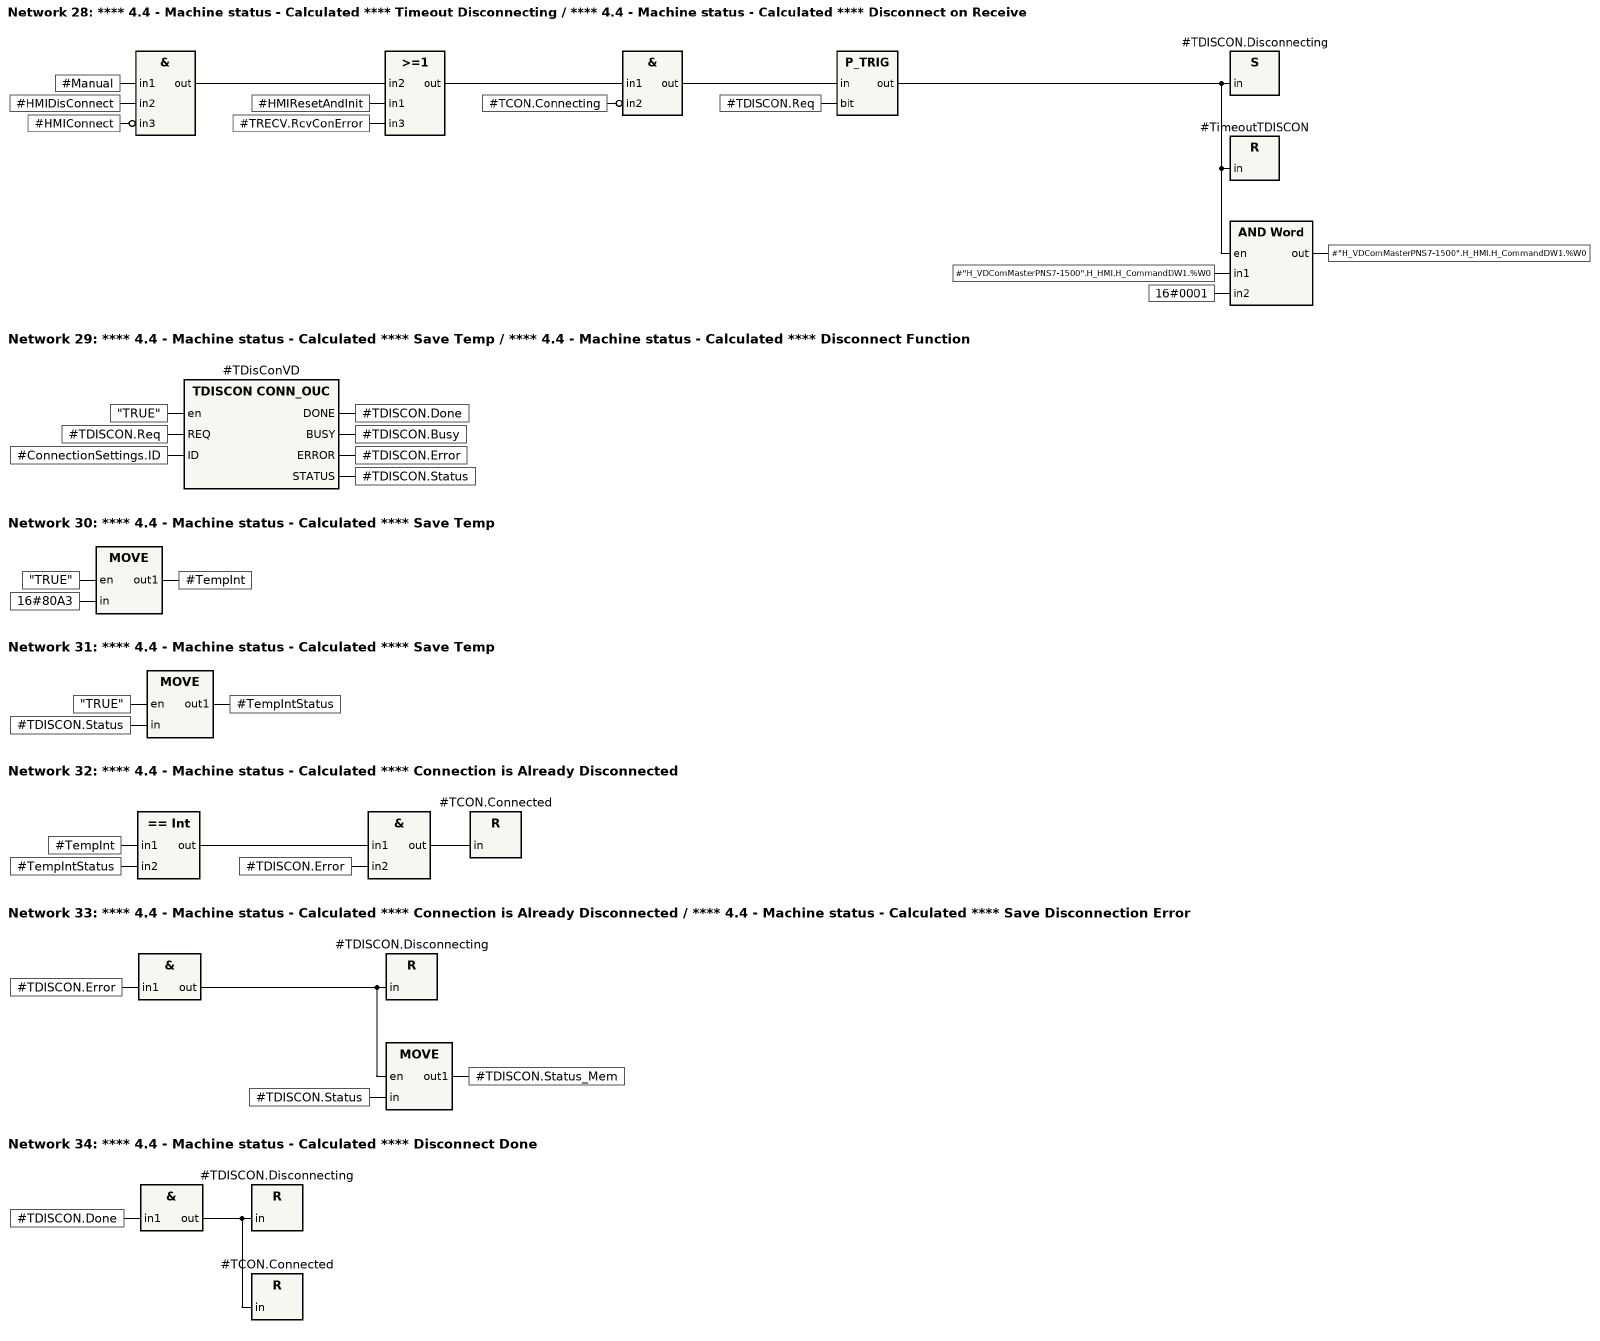
   #_w1 := ((#Manual AND #HMIDisConnect AND NOT #HMIConnect) OR #HMIResetAndInit OR #TRECV.RcvConError) AND NOT #TCON.Connecting;
   #_w2 := #_w1 AND NOT #TDISCON.Req;   // rising edge
   #TDISCON.Req := #_w1;
   IF #_w2 THEN
       #TDISCON.Disconnecting := TRUE;
       #TimeoutTDISCON := FALSE;
       #"H_VDComMasterPNS7-1500".H_HMI.H_CommandDW1.%W0 := #"H_VDComMasterPNS7-1500".H_HMI.H_CommandDW1.%W0 AND 16#0001;
   END_IF;
END_REGION

REGION Network 29: **** 4.4 - Machine status - Calculated **** Save Temp / **** 4.4 - Machine status - Calculated **** Disconnect Function
   // Temp / Disconnect function
   IF "TRUE" THEN
       #TDisConVD(REQ := #TDISCON.Req,   // TDISCON
                  ID := #ConnectionSettings.ID,
                  DONE => #TDISCON.Done,
                  BUSY => #TDISCON.Busy,
                  ERROR => #TDISCON.Error,
                  STATUS => #TDISCON.Status);
   END_IF;
END_REGION

REGION Network 30: **** 4.4 - Machine status - Calculated **** Save Temp
   // Temp
   IF "TRUE" THEN #TempInt := 16#80A3; END_IF;
END_REGION

REGION Network 31: **** 4.4 - Machine status - Calculated **** Save Temp
   // Temp
   IF "TRUE" THEN #TempIntStatus := #TDISCON.Status; END_IF;
END_REGION

REGION Network 32: **** 4.4 - Machine status - Calculated **** Connection is Already Disconnected
   // Connection is Already Disconnected
   IF (#TempInt = #TempIntStatus) AND #TDISCON.Error THEN #TCON.Connected := FALSE; END_IF;
END_REGION

REGION Network 33: **** 4.4 - Machine status - Calculated **** Connection is Already Disconnected / **** 4.4 - Machine status - Calculated **** Save Disconnection Error
   // Connection is Already Disconnected / Save Disconnection error
   IF #TDISCON.Error THEN
       #TDISCON.Disconnecting := FALSE;
       #TDISCON.Status_Mem := #TDISCON.Status;
   END_IF;
END_REGION

REGION Network 34: **** 4.4 - Machine status - Calculated **** Disconnect Done
   // Disconnect Done
   IF #TDISCON.Done THEN
       #TDISCON.Disconnecting := FALSE;
       #TCON.Connected := FALSE;
   END_IF;
END_REGION

REGION Network 35: **** 4.4 - Machine status - Calculated **** Diconnect / **** 4.4 - Machine status - Calculated **** Disconnect
   // Diconnect / Disconnect
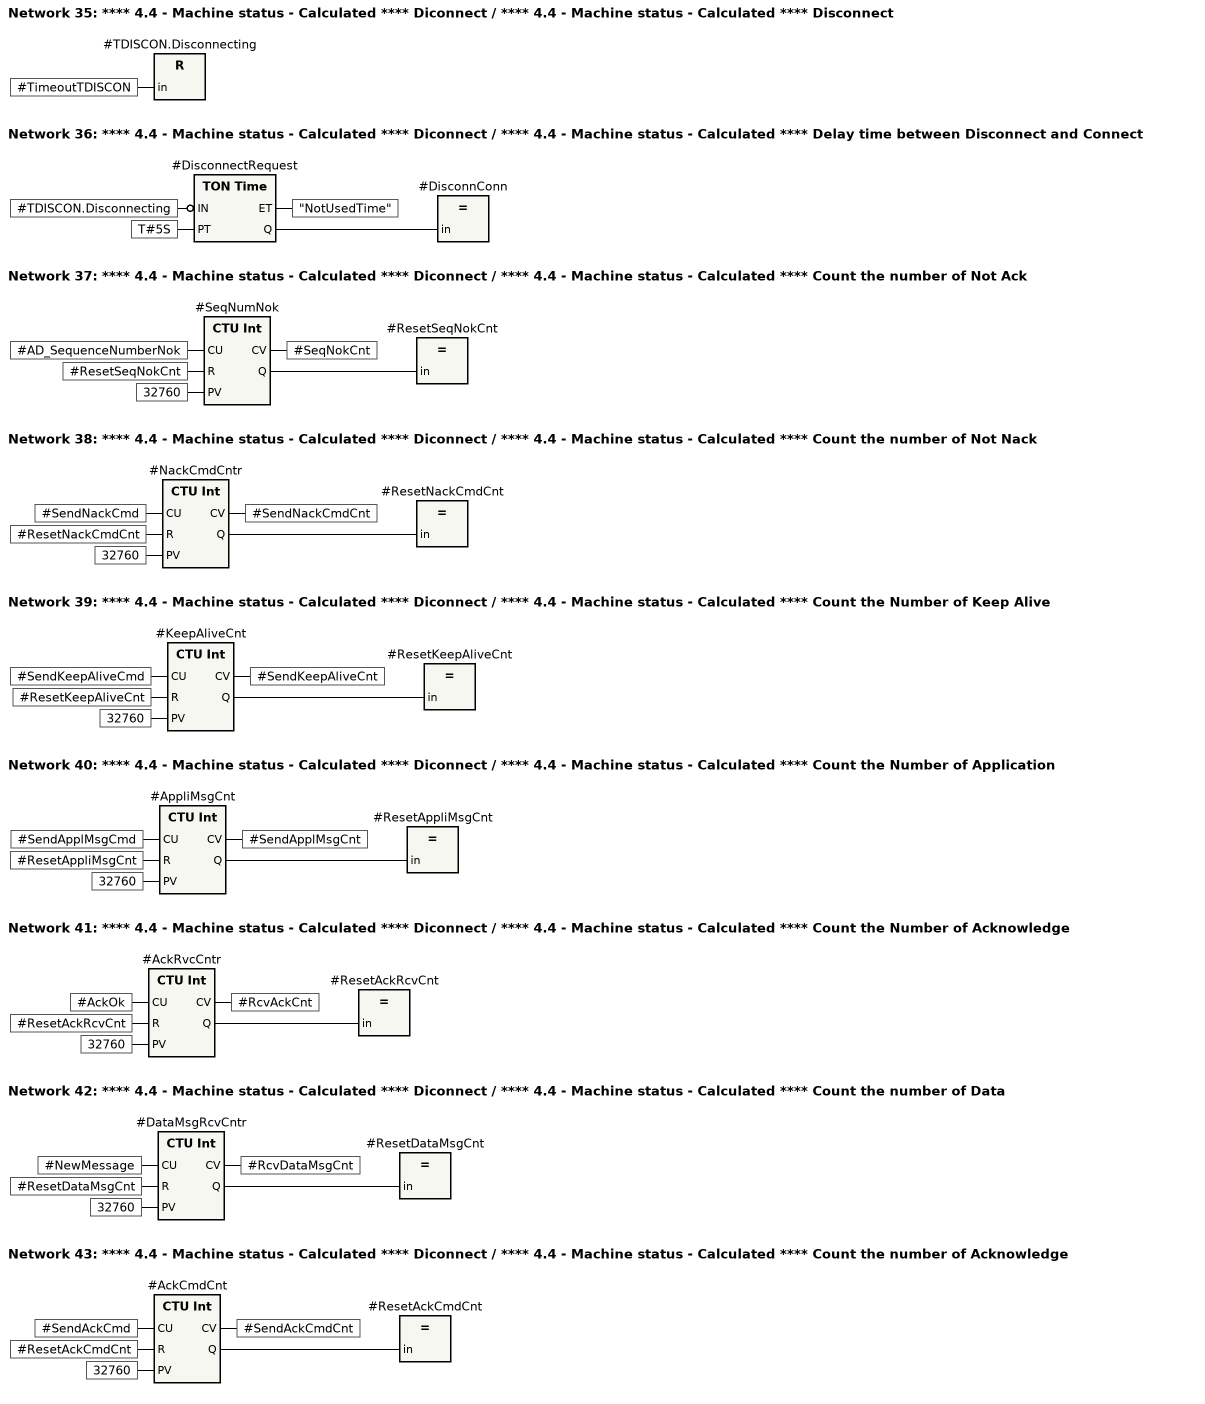
   IF #TimeoutTDISCON THEN #TDISCON.Disconnecting := FALSE; END_IF;
END_REGION

REGION Network 36: **** 4.4 - Machine status - Calculated **** Diconnect / **** 4.4 - Machine status - Calculated **** Delay time between Disconnect and Connect
   // Diconnect / Delay time between disconnect and connect
   #DisconnectRequest(IN := NOT #TDISCON.Disconnecting, PT := T#5S, ET => "NotUsedTime");   // TON
   #DisconnConn := #DisconnectRequest.Q;
END_REGION

REGION Network 37: **** 4.4 - Machine status - Calculated **** Diconnect / **** 4.4 - Machine status - Calculated **** Count the number of Not Ack
   // Diconnect / Count the number of Not acknowledge messages; for diagnostics only
   #SeqNumNok(CU := #AD_SequenceNumberNok, R := #ResetSeqNokCnt, PV := 32760, CV => #SeqNokCnt);   // CTU
   #ResetSeqNokCnt := #SeqNumNok.Q;
END_REGION

REGION Network 38: **** 4.4 - Machine status - Calculated **** Diconnect / **** 4.4 - Machine status - Calculated **** Count the number of Not Nack
   // Diconnect / Count the number of Not acknowledge messages; for diagnostics only
   #NackCmdCntr(CU := #SendNackCmd, R := #ResetNackCmdCnt, PV := 32760, CV => #SendNackCmdCnt);   // CTU
   #ResetNackCmdCnt := #NackCmdCntr.Q;
END_REGION

REGION Network 39: **** 4.4 - Machine status - Calculated **** Diconnect / **** 4.4 - Machine status - Calculated **** Count the Number of Keep Alive
   // Diconnect / Count the number of keep alive messages; for diagnostics only
   #KeepAliveCnt(CU := #SendKeepAliveCmd, R := #ResetKeepAliveCnt, PV := 32760, CV => #SendKeepAliveCnt);   // CTU
   #ResetKeepAliveCnt := #KeepAliveCnt.Q;
END_REGION

REGION Network 40: **** 4.4 - Machine status - Calculated **** Diconnect / **** 4.4 - Machine status - Calculated **** Count the Number of Application
   // Diconnect / Count the number of Application messages; for diagnostics only
   #AppliMsgCnt(CU := #SendApplMsgCmd, R := #ResetAppliMsgCnt, PV := 32760, CV => #SendApplMsgCnt);   // CTU
   #ResetAppliMsgCnt := #AppliMsgCnt.Q;
END_REGION

REGION Network 41: **** 4.4 - Machine status - Calculated **** Diconnect / **** 4.4 - Machine status - Calculated **** Count the Number of Acknowledge
   // Diconnect / Count the number of Acknowledge messages received; for diagnostics only
   #AckRvcCntr(CU := #AckOk, R := #ResetAckRcvCnt, PV := 32760, CV => #RcvAckCnt);   // CTU
   #ResetAckRcvCnt := #AckRvcCntr.Q;
END_REGION

REGION Network 42: **** 4.4 - Machine status - Calculated **** Diconnect / **** 4.4 - Machine status - Calculated **** Count the number of Data
   // Diconnect / Count the number of Data messages received; for diagnostics only
   #DataMsgRcvCntr(CU := #NewMessage, R := #ResetDataMsgCnt, PV := 32760, CV => #RcvDataMsgCnt);   // CTU
   #ResetDataMsgCnt := #DataMsgRcvCntr.Q;
END_REGION

REGION Network 43: **** 4.4 - Machine status - Calculated **** Diconnect / **** 4.4 - Machine status - Calculated **** Count the number of Acknowledge
   // Diconnect / Count the number of Acknowledge messages; for diagnostics only
   #AckCmdCnt(CU := #SendAckCmd, R := #ResetAckCmdCnt, PV := 32760, CV => #SendAckCmdCnt);   // CTU
   #ResetAckCmdCnt := #AckCmdCnt.Q;
END_REGION

NETWORK
TITLE = **** 4.4 - Machine status - Calculated **** Pointers
// Build the any pointers to the different DB's, needed for:
//  * BLKMOV (RecvPointer & BufferPointer)
//  * SEND (FB63 -> TSEND)
//  * RCV  (FB64 -> TRCV)
// Common Pointer parameters for
//  * RECV DB
//  * SEND DB
//  * SEND Buf DB
      LAR1  P##PointerRecv;
      L     16#1002;
      T     LW [AR1, P#0.0];
      LAR1  P##PointerSend;
      L     16#1002;
      T     LW [AR1, P#0.0];
      LAR1  P##PointerSendBuf;
      L     16#1002;
      T     LW [AR1, P#0.0];
// Cleaning Warnings APa
//      L     16#10                // S7  S7
//      T     %LB0                 // RECV
//      T     %LB10                // SEND
//      T     %LB20                // SEND BUF
//
//      L     16#02                //Data type (Bytes = 2)
//      T     %LB1                 // RECV
//      T     %LB11                // SEND
//      T     %LB21                // SEND BUF
      L     #RecvDBNbr;
      T     #RecvDBNO;

      CALL  ATTR_DB
      ( REQ       := "TRUE",
        DB_NUMBER := #RecvDBNO,
        RET_VAL   := "NotUsedInt",
        DB_LENGTH := #LengthDB,
        ATTRIB    := "NotUsedByte"
      );

//DB Header
      LAR1  P##PointerRecv;
      L     #LengthDB;
      T     LW [AR1, P#2.0];
      LAR1  P##PointerSend;
      L     16#000A;  //LengthLength
      T     LW [AR1, P#2.0];


//      L     #LengthDB
//      T     %LW2                 // RECV
//      L     16#000A              //LengthLength
//      T     %LW12                // SEND
      LAR1  P##PointerRecv;
      L     0;
      SLD   3;
      OD    16#8400_0000;
      T     LD [AR1, P#6.0];

      LAR1  P##PointerSend;
      L     0;
      SLD   3;
      OD    16#8400_0000;
      T     LD [AR1, P#6.0];


      LAR1  P##PointerSendBuf;
      L     0;
      SLD   3;
      OD    16#8400_0000;
      T     LD [AR1, P#6.0];

//      L     L#0                  //Offset in DB
//      SLD   3                    // Convert to pointer Convert to pointer
//      T     %LD6                 // RECV
//      T     %LD16                // SEND
//      T     %LD26                // SEND BUF

// Pointer to the Receive DB (Pointer_RECV) // DB no DB no
      LAR1  P##PointerRecv;
      L     #RecvDBNbr;
      T     LW [AR1, P#4.0];

//      L     #RecvDBNbr
//      T     %LW4                 // RECV

// Pointer to the Send DB (Pointer_SEND) Pointer to the Send DB (Pointer_SEND)
// DB no DB no
      LAR1  P##PointerSend;
      L     #SendDBNbr;
      T     LW [AR1, P#4.0];

//      L     #SendDBNbr
//      T     %LW14                // SEND

// Set memory area to DB Set memory area to DB
//      L     16#84                // Memory area DB Memory area DB
//      T     %LB6                 // RECV
//      T     %LB16                // SEND
//      T     %LB26                // SEND BUF




REGION Network 45: **** 4.4 - Machine status - Calculated **** Received Data
   // Received Data:
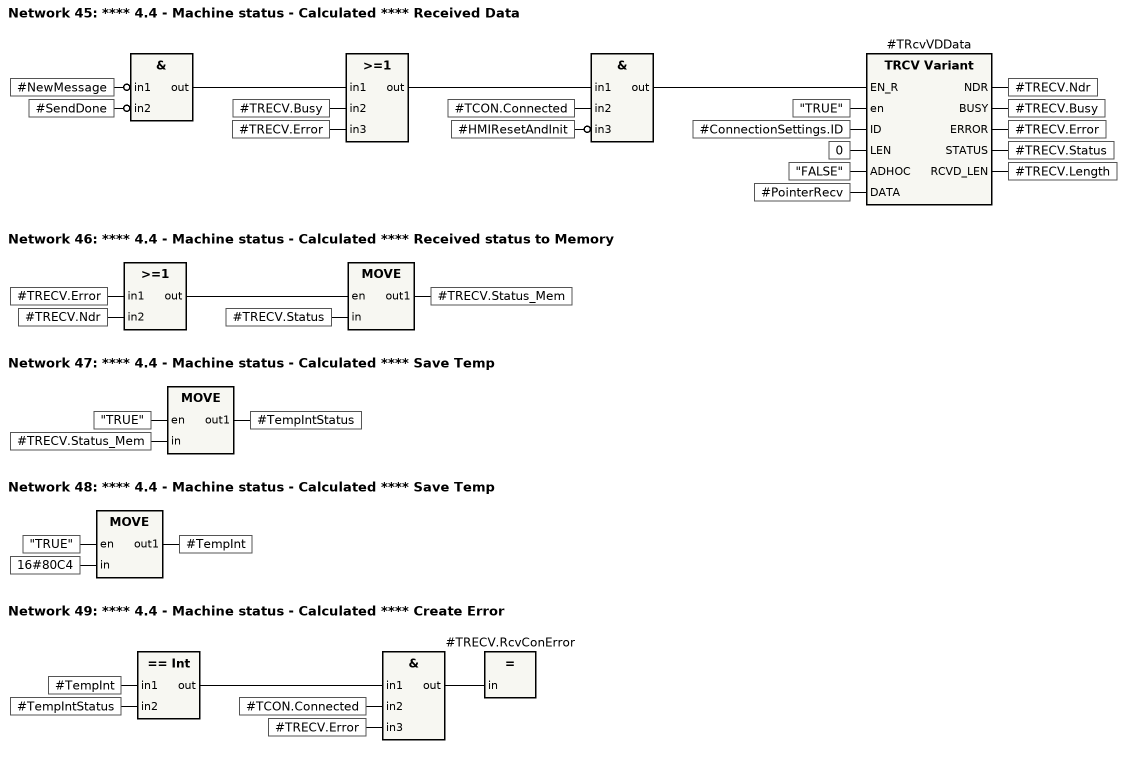
   IF "TRUE" THEN
       #TRcvVDData(EN_R := ((NOT #NewMessage AND NOT #SendDone) OR #TRECV.Busy OR #TRECV.Error) AND #TCON.Connected AND NOT #HMIResetAndInit,   // TRCV
                   ID := #ConnectionSettings.ID,
                   LEN := 0,
                   ADHOC := "FALSE",
                   DATA := #PointerRecv,
                   NDR => #TRECV.Ndr,
                   BUSY => #TRECV.Busy,
                   ERROR => #TRECV.Error,
                   STATUS => #TRECV.Status,
                   RCVD_LEN => #TRECV.Length);
   END_IF;
END_REGION

REGION Network 46: **** 4.4 - Machine status - Calculated **** Received status to Memory
   // Received status to memory
   IF #TRECV.Error OR #TRECV.Ndr THEN #TRECV.Status_Mem := #TRECV.Status; END_IF;
END_REGION

REGION Network 47: **** 4.4 - Machine status - Calculated **** Save Temp
   // Temp
   IF "TRUE" THEN #TempIntStatus := #TRECV.Status_Mem; END_IF;
END_REGION

REGION Network 48: **** 4.4 - Machine status - Calculated **** Save Temp
   // Temp
   IF "TRUE" THEN #TempInt := 16#80C4; END_IF;
END_REGION

REGION Network 49: **** 4.4 - Machine status - Calculated **** Create Error
   // Create error when status is equal to 0x80C4
   #TRECV.RcvConError := (#TempInt = #TempIntStatus) AND #TCON.Connected AND #TRECV.Error;
END_REGION

REGION Network 50: **** 4.6 - Machine Status - Indication **** Icon Animation
   // Icon Animation
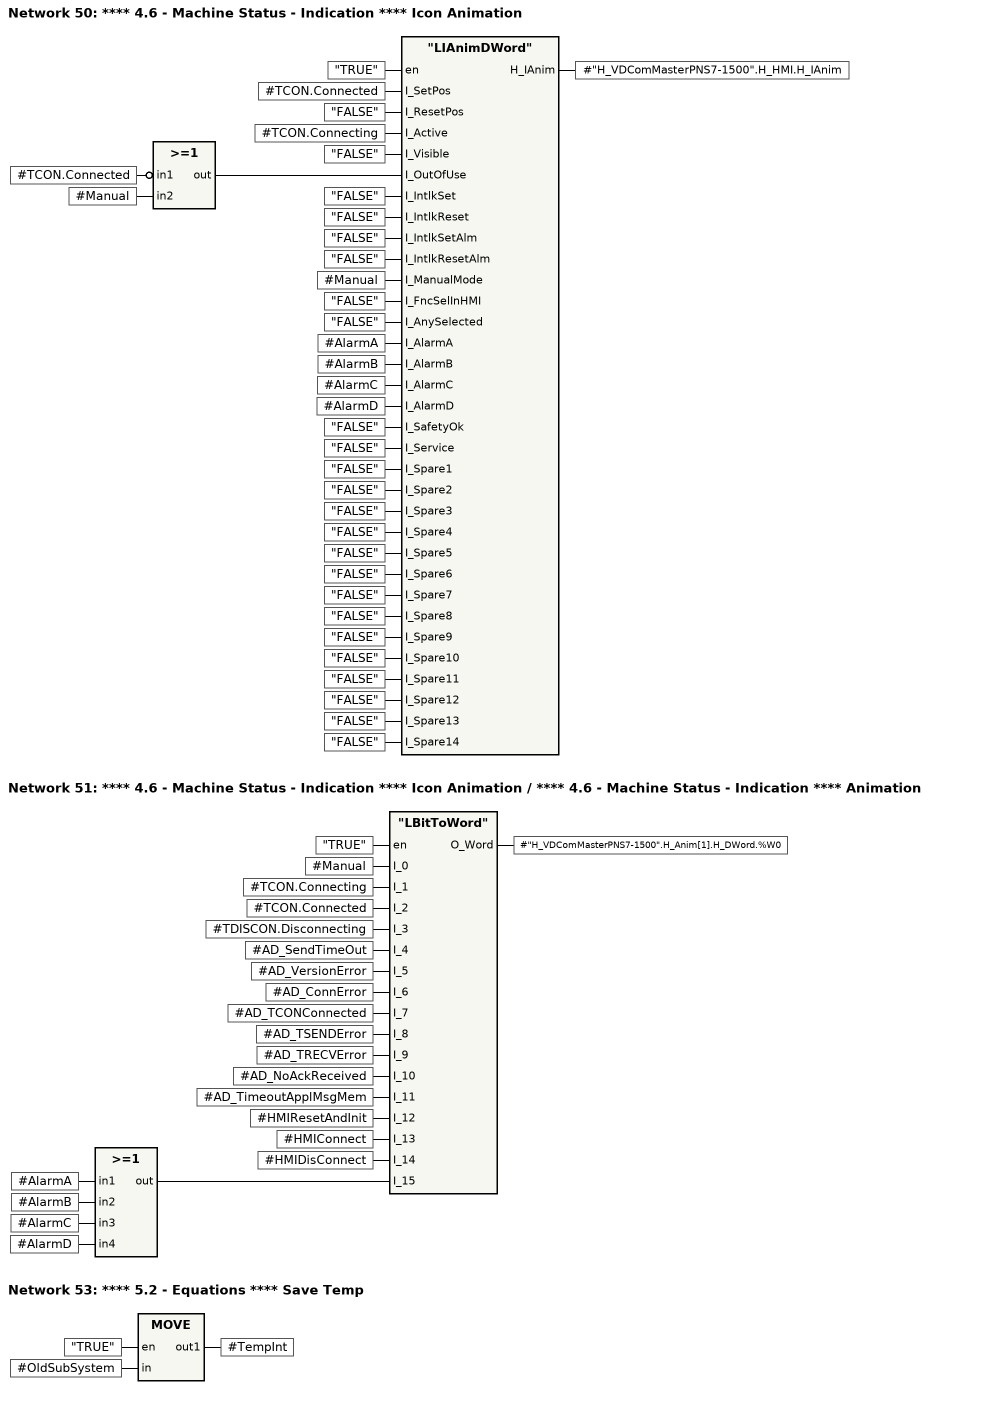
   IF "TRUE" THEN
       "LIAnimDWord"(I_SetPos := #TCON.Connected,
                     I_ResetPos := "FALSE",
                     I_Active := #TCON.Connecting,
                     I_Visible := "FALSE",
                     I_OutOfUse := NOT #TCON.Connected OR #Manual,
                     I_IntlkSet := "FALSE",
                     I_IntlkReset := "FALSE",
                     I_IntlkSetAlm := "FALSE",
                     I_IntlkResetAlm := "FALSE",
                     I_ManualMode := #Manual,
                     I_FncSelInHMI := "FALSE",
                     I_AnySelected := "FALSE",
                     I_AlarmA := #AlarmA,
                     I_AlarmB := #AlarmB,
                     I_AlarmC := #AlarmC,
                     I_AlarmD := #AlarmD,
                     I_SafetyOk := "FALSE",
                     I_Service := "FALSE",
                     I_Spare1 := "FALSE",
                     I_Spare2 := "FALSE",
                     I_Spare3 := "FALSE",
                     I_Spare4 := "FALSE",
                     I_Spare5 := "FALSE",
                     I_Spare6 := "FALSE",
                     I_Spare7 := "FALSE",
                     I_Spare8 := "FALSE",
                     I_Spare9 := "FALSE",
                     I_Spare10 := "FALSE",
                     I_Spare11 := "FALSE",
                     I_Spare12 := "FALSE",
                     I_Spare13 := "FALSE",
                     I_Spare14 := "FALSE",
                     H_IAnim => #"H_VDComMasterPNS7-1500".H_HMI.H_IAnim);
   END_IF;
END_REGION

REGION Network 51: **** 4.6 - Machine Status - Indication **** Icon Animation / **** 4.6 - Machine Status - Indication **** Animation
   // Icon Animation / Animation
   IF "TRUE" THEN
       "LBitToWord"(I_0 := #Manual,
                    I_1 := #TCON.Connecting,
                    I_2 := #TCON.Connected,
                    I_3 := #TDISCON.Disconnecting,
                    I_4 := #AD_SendTimeOut,
                    I_5 := #AD_VersionError,
                    I_6 := #AD_ConnError,
                    I_7 := #AD_TCONConnected,
                    I_8 := #AD_TSENDError,
                    I_9 := #AD_TRECVError,
                    I_10 := #AD_NoAckReceived,
                    I_11 := #AD_TimeoutApplMsgMem,
                    I_12 := #HMIResetAndInit,
                    I_13 := #HMIConnect,
                    I_14 := #HMIDisConnect,
                    I_15 := #AlarmA OR #AlarmB OR #AlarmC OR #AlarmD,
                    O_Word => #"H_VDComMasterPNS7-1500".H_Anim[1].H_DWord.%W0);
   END_IF;
END_REGION

NETWORK
TITLE = **** 5.2 - Equations **** MessageType to Local Variable
// Check that the received data is Ok Copy MessageType to local variable
      OPN   #I_VDCommRecvDB;
      L     %DBW0;  // VDVersion must always be same
      L     16#0100;
      <>I;
      =     #AD_VersionError;

      L     16#0100;
      T     %DBW0;

// Check new SeqNbr
      A     #TRECV.Ndr;  // New data is received
      A(;
      O(;
      L     %DBW8;  // Check seq nbr Ok
      L     #OldRecMsgNbr;
      <>I;
      );
      O(;
      L     %DBW8;  // Check seq nbr Ok
      L     0;
      ==I;
      );
      );
      S     #NewMsgNbr;

//-----------------------------------------------------------
// For next cycle OldRecSeqNbr=0 NewSeqNbr will always be Ok
//      L     -1
//      T     #OldRecMsgNbr
//-----------------------------------------------------------

// Check Messagetype
      L     %DBW4;
      L     2;
      >I;
      =     #UserMsgType;  // Messagetype > 2 then Ok message
      AN    #UserMsgType;
      JC    RSEQ;
//Remember messagenumber
      L     %DBW8;
      T     #OldRecMsgNbr;  // Remember last seq nbr
      L     %DBW6;
      T     #OldSubSystem;  // Remember last subsystem
RSEQ: NOP   0;

// Ack recieved Ack recieved
      L     %DBW4;
      L     1;
      ==I;
      =     #AckRcvd;

      L     %DBW8;
      L     #SendMsgNbr;
      ==I;
      =     #SeqNbrOk;  // Sequence number Ok for Ack rcvd

// Message length
      L     %DBW2;  // Message length in DB_RECV
      T     #MessageLengthRecv;

// Sequence number NOK
      A     #TRECV.Ndr;  // New data is received
      A     #UserMsgType;  // Data is of User type
      AN    #NewMsgNbr;  // Sequence number is NOK
      O     #AD_SequenceNumberNok;  // Hold status
      AN    #NewMsgNbr;  // Sequence number is NOK
      =     #AD_SequenceNumberNok;  // Sequence number NOK



REGION Network 53: **** 5.2 - Equations **** Save Temp
   // Temp
   IF "TRUE" THEN #TempInt := #OldSubSystem; END_IF;
END_REGION

REGION Network 54: **** 5.2 - Equations **** Receive Length
   // Receive length only copy if Ndr of read is set to 1
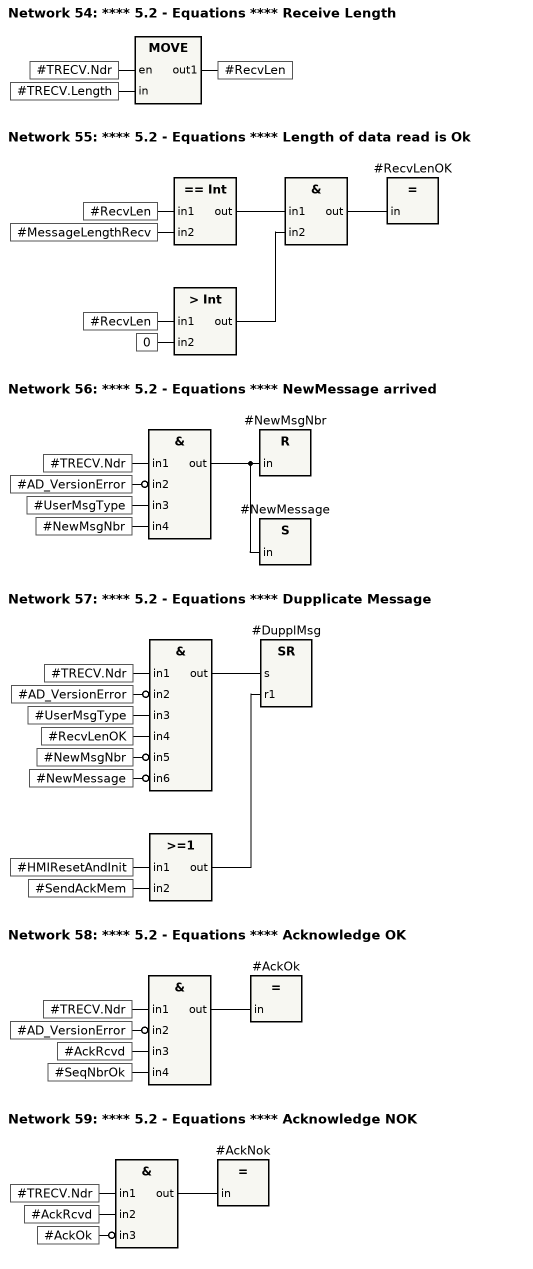
   IF #TRECV.Ndr THEN #RecvLen := #TRECV.Length; END_IF;
END_REGION

REGION Network 55: **** 5.2 - Equations **** Length of data read is Ok
   // Length of data read is Ok
   #RecvLenOK := (#RecvLen = #MessageLengthRecv) AND (#RecvLen > 0);
END_REGION

REGION Network 56: **** 5.2 - Equations **** NewMessage arrived
   // If new data is available and the data is Ok, then set output to subsystems NewMessage arrived.
   #_w1 := #TRECV.Ndr AND NOT #AD_VersionError AND #UserMsgType AND #NewMsgNbr;
   IF #_w1 THEN
       #NewMsgNbr := FALSE;
       #NewMessage := TRUE;
   END_IF;
END_REGION

REGION Network 57: **** 5.2 - Equations **** Dupplicate Message
   // Dupplicate Message
   IF #TRECV.Ndr AND NOT #AD_VersionError AND #UserMsgType AND #RecvLenOK AND NOT #NewMsgNbr AND NOT #NewMessage THEN
       #DupplMsg := TRUE;   // SR flip-flop
   END_IF;
   IF #HMIResetAndInit OR #SendAckMem THEN #DupplMsg := FALSE; END_IF;
END_REGION

REGION Network 58: **** 5.2 - Equations **** Acknowledge OK
   // Acknowledge OK
   #AckOk := #TRECV.Ndr AND NOT #AD_VersionError AND #AckRcvd AND #SeqNbrOk;
END_REGION

REGION Network 59: **** 5.2 - Equations **** Acknowledge NOK
   // Acknowledge not OK
   #AckNok := #TRECV.Ndr AND #AckRcvd AND NOT #AckOk;
END_REGION

REGION Network 60: **** 7.2 - Submodules - Command **** Postpone Send Ack
   // Time to postpone to send Ack upon reception of new message. This to prevent thatmessages are send too fast.
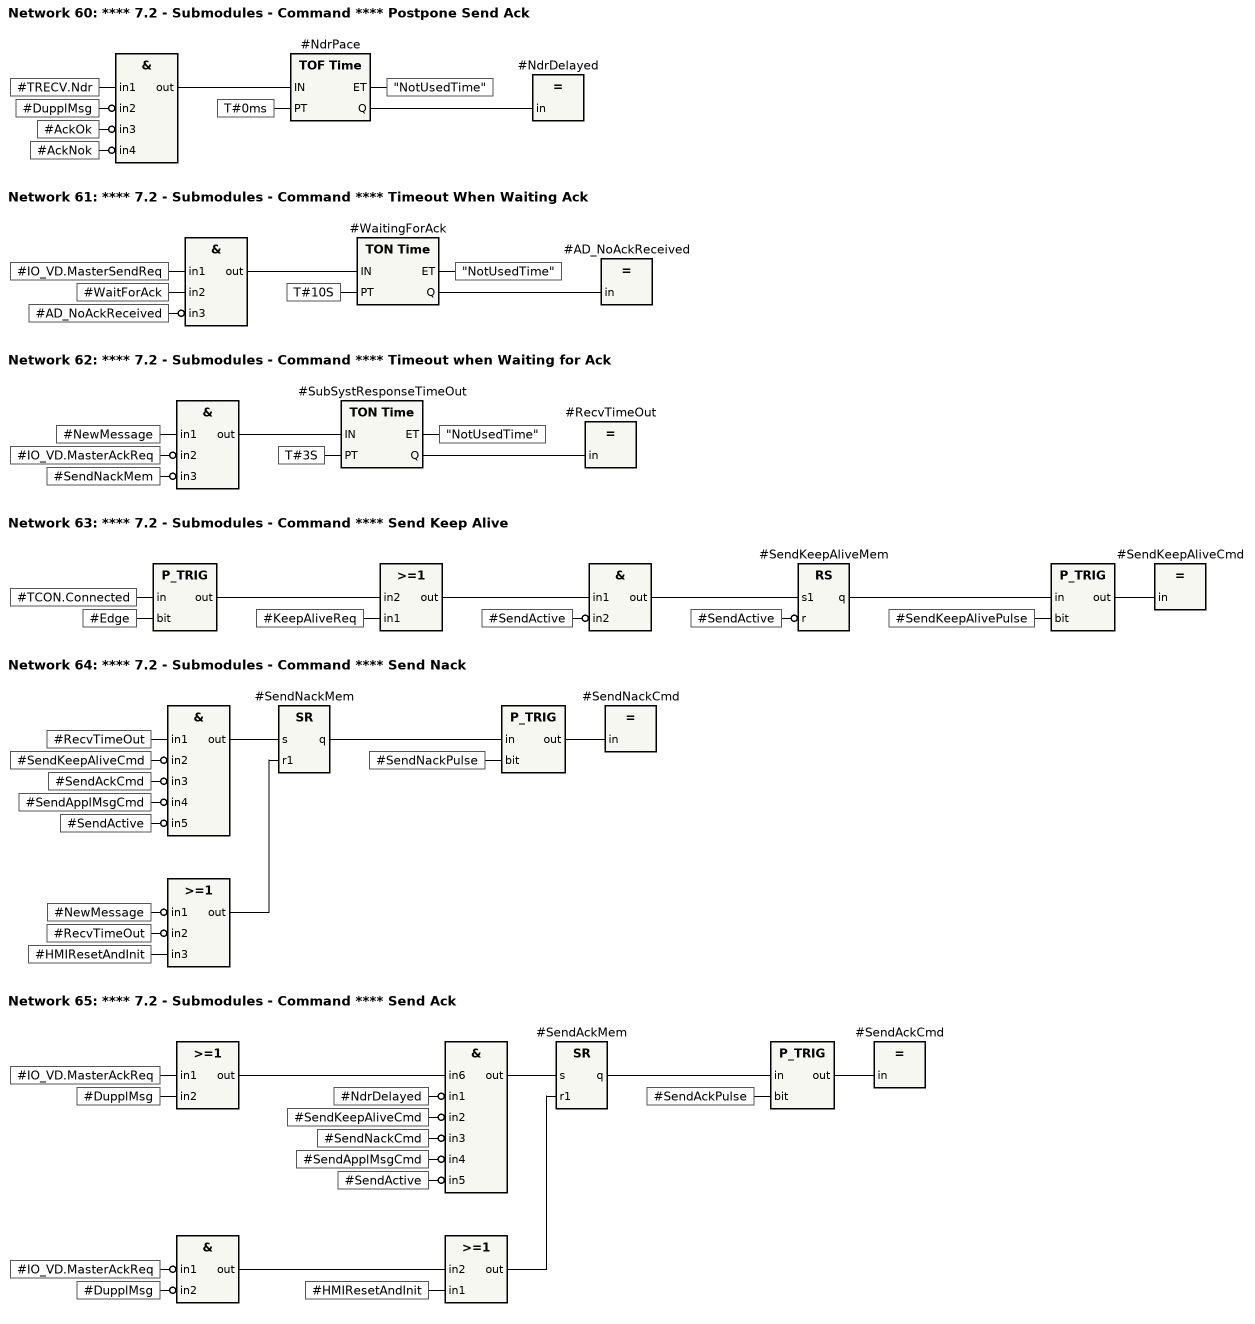
   #NdrPace(IN := #TRECV.Ndr AND NOT #DupplMsg AND NOT #AckOk AND NOT #AckNok, PT := T#0ms, ET => "NotUsedTime");   // TOF
   #NdrDelayed := #NdrPace.Q;
END_REGION

REGION Network 61: **** 7.2 - Submodules - Command **** Timeout When Waiting Ack
   // Timeout when waiting for Ack from superior system
   #WaitingForAck(IN := #IO_VD.MasterSendReq AND #WaitForAck AND NOT #AD_NoAckReceived,   // TON
                  PT := T#10S,
                  ET => "NotUsedTime");
   #AD_NoAckReceived := #WaitingForAck.Q;
END_REGION

REGION Network 62: **** 7.2 - Submodules - Command **** Timeout when Waiting for Ack
   // Timeout when waiting for Acknowlegde Request from Subsystem
   #SubSystResponseTimeOut(IN := #NewMessage AND NOT #IO_VD.MasterAckReq AND NOT #SendNackMem,   // TON
                           PT := T#3S,
                           ET => "NotUsedTime");
   #RecvTimeOut := #SubSystResponseTimeOut.Q;
END_REGION

REGION Network 63: **** 7.2 - Submodules - Command **** Send Keep Alive
   // Send Keep Alive
   #_w1 := #TCON.Connected AND NOT #Edge;   // rising edge
   #Edge := #TCON.Connected;
   IF NOT #SendActive THEN
       #SendKeepAliveMem := FALSE;   // RS flip-flop
   END_IF;
   IF (#_w1 OR #KeepAliveReq) AND NOT #SendActive THEN #SendKeepAliveMem := TRUE; END_IF;
   #_w2 := #SendKeepAliveMem AND NOT #SendKeepAlivePulse;   // rising edge
   #SendKeepAlivePulse := #SendKeepAliveMem;
   #SendKeepAliveCmd := #_w2;
END_REGION

REGION Network 64: **** 7.2 - Submodules - Command **** Send Nack
   // Send Nack when no subsystem is reacting on a new message received. This means 
   // that the new messages was not recognised by one of the subsystems ( subsystem 
   // number wrong or Messagetype wrong). Then the sender should be aware that what 
   // was send has no client.
   IF #RecvTimeOut AND NOT #SendKeepAliveCmd AND NOT #SendAckCmd AND NOT #SendApplMsgCmd AND NOT #SendActive THEN
       #SendNackMem := TRUE;   // SR flip-flop
   END_IF;
   IF NOT #NewMessage OR NOT #RecvTimeOut OR #HMIResetAndInit THEN #SendNackMem := FALSE; END_IF;
   #_w1 := #SendNackMem AND NOT #SendNackPulse;   // rising edge
   #SendNackPulse := #SendNackMem;
   #SendNackCmd := #_w1;
END_REGION

REGION Network 65: **** 7.2 - Submodules - Command **** Send Ack
   // Send Ack
   IF (#IO_VD.MasterAckReq OR #DupplMsg) AND NOT #NdrDelayed AND NOT #SendKeepAliveCmd AND NOT #SendNackCmd AND NOT #SendApplMsgCmd AND NOT #SendActive THEN
       #SendAckMem := TRUE;   // SR flip-flop
   END_IF;
   IF (NOT #IO_VD.MasterAckReq AND NOT #DupplMsg) OR #HMIResetAndInit THEN #SendAckMem := FALSE; END_IF;
   #_w1 := #SendAckMem AND NOT #SendAckPulse;   // rising edge
   #SendAckPulse := #SendAckMem;
   #SendAckCmd := #_w1;
END_REGION

REGION Network 66: **** 7.2 - Submodules - Command **** Ack Nack Sent
   // Ack Nack Sent
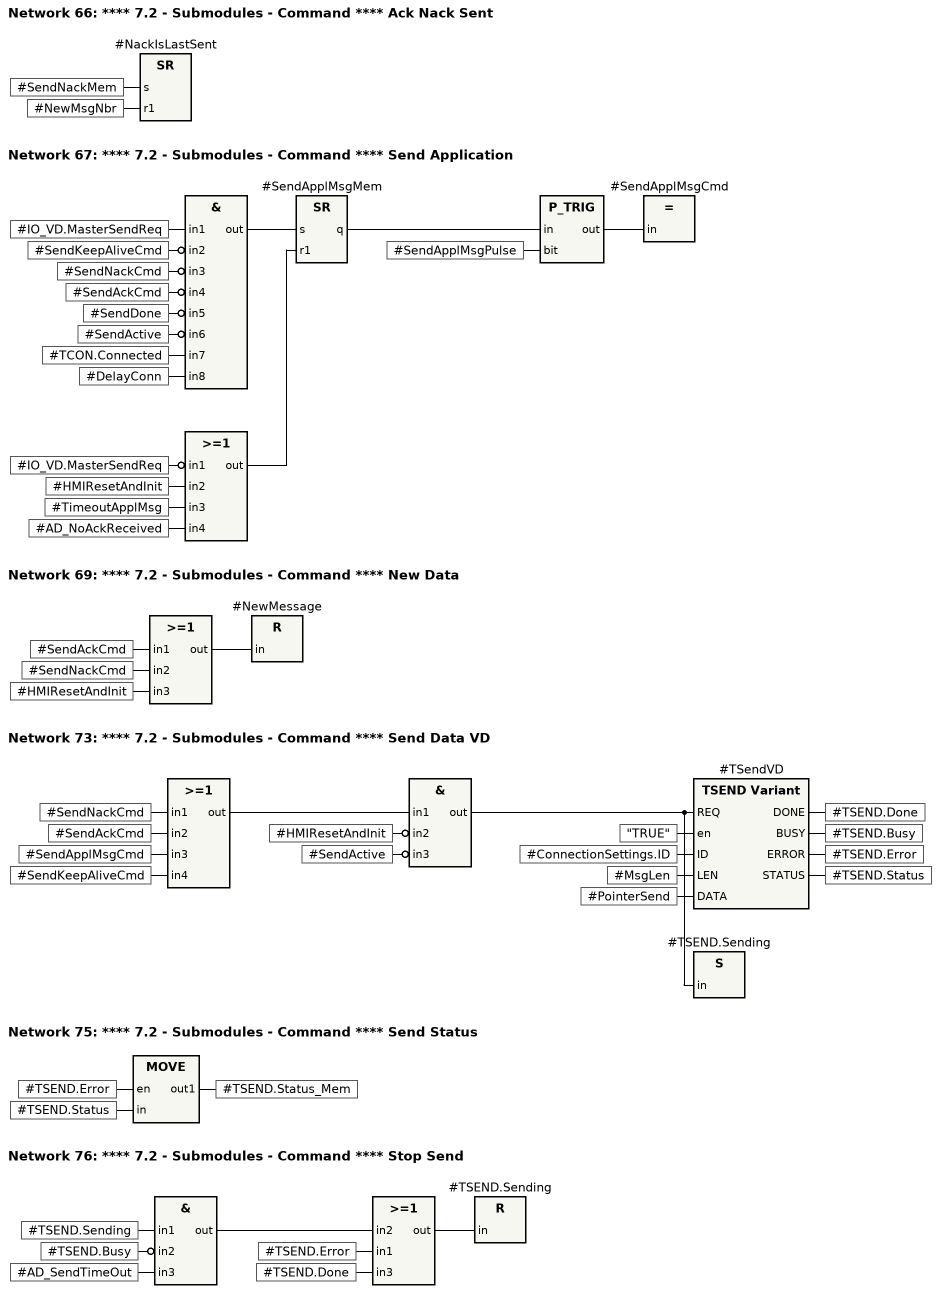
   IF #SendNackMem THEN
       #NackIsLastSent := TRUE;   // SR flip-flop
   END_IF;
   IF #NewMsgNbr THEN #NackIsLastSent := FALSE; END_IF;
END_REGION

REGION Network 67: **** 7.2 - Submodules - Command **** Send Application
   // Send Application
   IF #IO_VD.MasterSendReq AND NOT #SendKeepAliveCmd AND NOT #SendNackCmd AND NOT #SendAckCmd AND NOT #SendDone AND NOT #SendActive AND #TCON.Connected AND #DelayConn THEN
       #SendApplMsgMem := TRUE;   // SR flip-flop
   END_IF;
   IF NOT #IO_VD.MasterSendReq OR #HMIResetAndInit OR #TimeoutApplMsg OR #AD_NoAckReceived THEN
       #SendApplMsgMem := FALSE;
   END_IF;
   #_w1 := #SendApplMsgMem AND NOT #SendApplMsgPulse;   // rising edge
   #SendApplMsgPulse := #SendApplMsgMem;
   #SendApplMsgCmd := #_w1;
END_REGION

NETWORK
TITLE = **** 7.2 - Submodules - Command **** Send Application Sub System
// Send Application Sub System
      A     #SendApplMsgCmd;
      JCN   nOZE;
      OPN   #IO_VD.VDCommSendDB;
      L     %DBW6;
      T     #"H_VDComMasterPNS7-1500".H_Anim[2].H_DWord.%W0;
nOZE: NOP   0;


REGION Network 69: **** 7.2 - Submodules - Command **** New Data
   // If New Data is Available And the data is Ok, then set output to subsystems
   IF #SendAckCmd OR #SendNackCmd OR #HMIResetAndInit THEN #NewMessage := FALSE; END_IF;
END_REGION

NETWORK
TITLE = **** 7.2 - Submodules - Command **** Keep Alive
// Keep Alive command
      A     #SendKeepAliveCmd;
      JCN   SKAC;
      OPN   #I_VDCommSendDB;
      L     10;  //LengthLength
      T     %DBW2;
      L     2;  // MessageTypeMessageType
      T     %DBW4;
      L     0;  // Subsystem
      T     %DBW6;
      L     0;  // MessageNumber (SeqNbr)
      T     %DBW8;
SKAC: NOP   0;


NETWORK
TITLE = **** 7.2 - Submodules - Command **** Check Received
// Check Received Data
      AN    #SendAckCmd;  // Send AckCmd
      JC    SACK;
      L     #OldRecMsgNbr;  // MessageNumber (SeqNbr)
      OPN   #I_VDCommSendDB;
      T     %DBW8;
      L     #OldSubSystem;  // Subsystem
      T     %DBW6;
      L     1;  // MessageType
      T     %DBW4;
      L     10;  //LengthLength
      T     %DBW2;
      JU    PAPM;
SACK: NOP   0;

      AN    #SendNackCmd;  // Send NackCmd
      JC    SNAC;
      L     #OldRecMsgNbr;  // MessageNumber (SeqNbr)
      OPN   #I_VDCommSendDB;
      T     %DBW8;
      L     #OldSubSystem;  // Subsystem
      T     %DBW6;
      L     0;  // MessageType
      T     %DBW4;
      L     10;  //LengthLength
      T     %DBW2;
      JU    PAPM;
SNAC: NOP   0;

      A     #SendApplMsgCmd;  // Send Application Message
      AN    #SendActive;
      AN    #SendDone;
      JCN   PAPM;

// Number of bytes to copy***************************************************************************************************
//     L     #I_VDCommSendDBBuf   // SEND BUF        APa Fixa S7-1500
//     T     #SS_Out_Buf          // DB number to copy
//     OPN DB [ #SS_Out_Buf]      // APa Fixa S7-1500
//     OPN   #I_VDCommSendDBBuf

      L     #IO_VD.VDCommSendDBNr;
      L     0;
      ==I;
//     JCN   NSrS1
      OPN   #IO_VD.VDCommSendDB;
      L     DBNO;
      T     #OutBuf;
      OPN   #IO_VD.VDCommSendDB;
      LAR1  P##PointerSendBuf;
      L     %DBW2;  // Length
      T     LW [AR1, P#2.0];
      OPN   #IO_VD.VDCommSendDB;
      LAR1  P##PointerSend;
      L     %DBW2;
      T     LW [AR1, P#2.0];
      OPN   #IO_VD.VDCommSendDB;
      L     DBNO;
      T     #OutBuf;
//NSrS1: NOP 0

//      OPN   #I_VDCommSendBufStn2 APa Fixa S7-1500
//    L DBNO
//   L     #I_VDCommSendDBBuf
//    ==I
//    L DBNO
//     T     #SS_Out_Buf
//     JCN   NSrS2
//      OPN   #I_VDCommSendBufStn2
//    L     %DBW2                // Length
//    T     %LW22                // SEND BUF
//     T     %LW12                // SEND
//     L DBNO
//      T     #SS_Out_Buf
//NSrS2: NOP 0

//*****************************************************************************************************************************


// Pointer to the Receive DB (Pointer_SEND_Buf) APa Fixa S7-1500
// DB no DB no
//    L DBNO
//  T     #SS_Out_Buf
//   L     #I_VDCommSendDBBuf
      OPN   #IO_VD.VDCommSendDB;
      L     DBNO;
      T     #OutBuf;
      L     #OutBuf;
      LAR1  P##PointerSendBuf;
      L     #OutBuf;
      T     LW [AR1, P#4.0];
//      T     %LW24                // SEND BUF
      CALL  BLKMOV
      ( SRCBLK  := #PointerSendBuf,  // SEND Buffer
        RET_VAL := "NotUsedInt",
        DSTBLK  := #PointerSend  // SEND
      );  // Copy data from buffer DB to send DB

      L     #SendMsgNbr;
      L     1000;
      >=I;
      JCN   ZermMsgCnt;
      L     1;
      T     #SendMsgNbr;

ZermMsgCnt:OPN   #I_VDCommSendDB;
      L     #SendMsgNbr;
      A     #AD_TimeoutApplMsgMem;
      JC    noin;
      L     #SendMsgNbr;
      +     1;
noin: T     #SendMsgNbr;
      T     %DBW8;  // Messagenumber

      CLR;
      R     #AD_TimeoutApplMsgMem;

PAPM: OPN   #I_VDCommSendDB;
      L     %DBW2;
      T     #MsgLen;

      L     1;
      T     %DBB0;

      A     #NackIsLastSent;
      A     #SendAckCmd;
      JCN   ZeroMesag;
      L     0;
      T     %DBW4;
ZeroMesag:NOP   0;

      L     #SendMsgNbr;
      T     "NotUsedDInt";

NETWORK
TITLE = **** 7.2 - Submodules - Command **** Length to Send Pointers
// Length to Send Pointers / Check Received Data
      LAR1  P##PointerSend;
      L     #MsgLen;
      T     LW [AR1, P#2.0];


REGION Network 73: **** 7.2 - Submodules - Command **** Send Data VD
   // Send Data VD
   #_w1 := (#SendNackCmd OR #SendAckCmd OR #SendApplMsgCmd OR #SendKeepAliveCmd) AND NOT #HMIResetAndInit AND NOT #SendActive;
   IF "TRUE" THEN
       #TSendVD(REQ := #_w1,   // TSEND
                ID := #ConnectionSettings.ID,
                LEN := #MsgLen,
                DATA := #PointerSend,
                DONE => #TSEND.Done,
                BUSY => #TSEND.Busy,
                ERROR => #TSEND.Error,
                STATUS => #TSEND.Status);
   END_IF;
   IF #_w1 THEN #TSEND.Sending := TRUE; END_IF;
END_REGION

NETWORK
TITLE = **** 7.2 - Submodules - Command **** Send Data to VD
// Send data to VD (length is the length in the SEND_DB)
      L     #TSEND.Status;
      L     16#0000;
      ==I;
      =     #SendJobCompleted;  // Send job completed without error
      L     #TSEND.Status;
      L     16#7000;
      ==I;
      =     #SendInactive;  // No job processing active
      L     #TSEND.Status;
      L     16#7001;
      ==I;
      =     #SendStartOfProc;  // Start of job processing, data being sent
      L     #TSEND.Status;
      L     16#7002;
      ==I;
      =     #SendFollowOnCall;  // Follow-on call (REQ irrelevant ), job being processed



REGION Network 75: **** 7.2 - Submodules - Command **** Send Status
   // Send Status to memory
   IF #TSEND.Error THEN #TSEND.Status_Mem := #TSEND.Status; END_IF;
END_REGION

REGION Network 76: **** 7.2 - Submodules - Command **** Stop Send
   // Stop sending  Error,Done,Sending AND NOT Busy
   IF (#TSEND.Sending AND NOT #TSEND.Busy AND #AD_SendTimeOut) OR #TSEND.Error OR #TSEND.Done THEN
       #TSEND.Sending := FALSE;
   END_IF;
END_REGION

REGION Network 77: **** 7.2 - Submodules - Command **** Send Active
   // Send Active
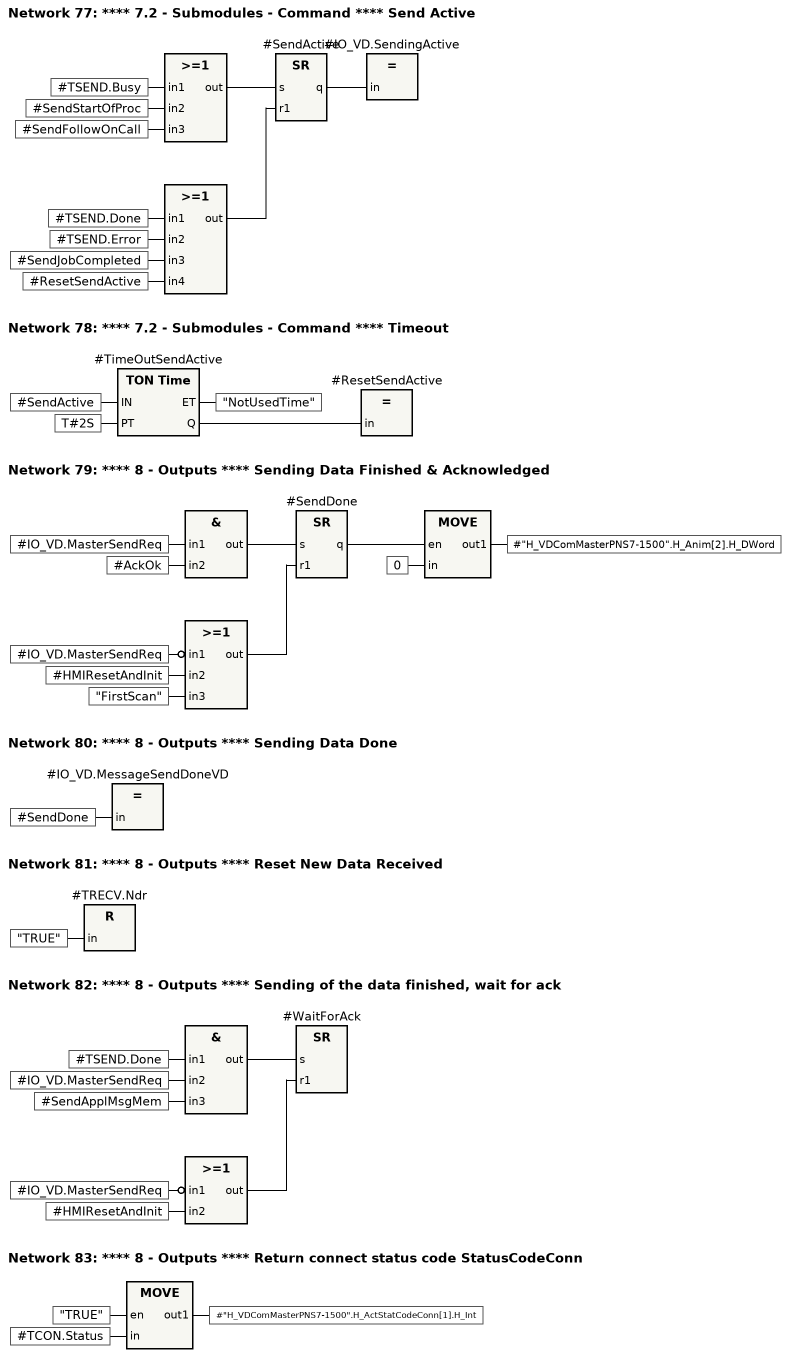
   IF #TSEND.Busy OR #SendStartOfProc OR #SendFollowOnCall THEN
       #SendActive := TRUE;   // SR flip-flop
   END_IF;
   IF #TSEND.Done OR #TSEND.Error OR #SendJobCompleted OR #ResetSendActive THEN #SendActive := FALSE; END_IF;
   #IO_VD.SendingActive := #SendActive;
END_REGION

REGION Network 78: **** 7.2 - Submodules - Command **** Timeout
   // Timeout
   #TimeOutSendActive(IN := #SendActive, PT := T#2S, ET => "NotUsedTime");   // TON
   #ResetSendActive := #TimeOutSendActive.Q;
END_REGION

REGION Network 79: **** 8 - Outputs **** Sending Data Finished & Acknowledged
   // Sending Data Finished & Acknowledged
   IF #IO_VD.MasterSendReq AND #AckOk THEN
       #SendDone := TRUE;   // SR flip-flop
   END_IF;
   IF NOT #IO_VD.MasterSendReq OR #HMIResetAndInit OR "FirstScan" THEN #SendDone := FALSE; END_IF;
   IF #SendDone THEN #"H_VDComMasterPNS7-1500".H_Anim[2].H_DWord := 0; END_IF;
END_REGION

REGION Network 80: **** 8 - Outputs **** Sending Data Done
   // Sending Data Done
   #IO_VD.MessageSendDoneVD := #SendDone;
END_REGION

REGION Network 81: **** 8 - Outputs **** Reset New Data Received
   // Reset "New data received" bit. All processing shall be done before this step.
   IF "TRUE" THEN #TRECV.Ndr := FALSE; END_IF;
END_REGION

REGION Network 82: **** 8 - Outputs **** Sending of the data finished, wait for ack
   // Sending of the data finished, wait for ack
   IF #TSEND.Done AND #IO_VD.MasterSendReq AND #SendApplMsgMem THEN
       #WaitForAck := TRUE;   // SR flip-flop
   END_IF;
   IF NOT #IO_VD.MasterSendReq OR #HMIResetAndInit THEN #WaitForAck := FALSE; END_IF;
END_REGION

REGION Network 83: **** 8 - Outputs **** Return connect status code StatusCodeConn
   // Return connect status code H_StatusCodeConn
   IF "TRUE" THEN #"H_VDComMasterPNS7-1500".H_ActStatCodeConn[1].H_Int := #TCON.Status; END_IF;
END_REGION

REGION Network 84: **** 8 - Outputs **** Return receive status code StatusCodeDisconn
   // Return receive status code H_StatusCodeDisconn
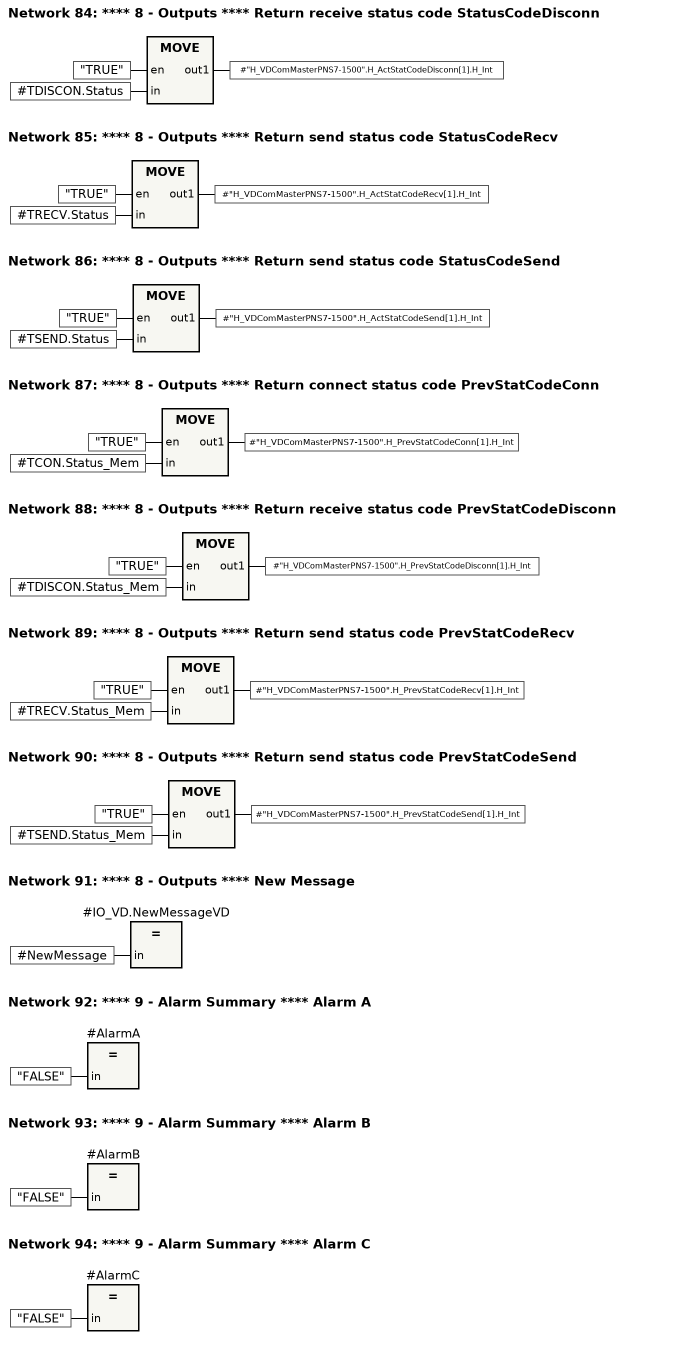
   IF "TRUE" THEN #"H_VDComMasterPNS7-1500".H_ActStatCodeDisconn[1].H_Int := #TDISCON.Status; END_IF;
END_REGION

REGION Network 85: **** 8 - Outputs **** Return send status code StatusCodeRecv
   // Return send status code H_StatusCodeRecv
   IF "TRUE" THEN #"H_VDComMasterPNS7-1500".H_ActStatCodeRecv[1].H_Int := #TRECV.Status; END_IF;
END_REGION

REGION Network 86: **** 8 - Outputs **** Return send status code StatusCodeSend
   // Return send status code H_StatusCodeSend
   IF "TRUE" THEN #"H_VDComMasterPNS7-1500".H_ActStatCodeSend[1].H_Int := #TSEND.Status; END_IF;
END_REGION

REGION Network 87: **** 8 - Outputs **** Return connect status code PrevStatCodeConn
   // Return connect status code H_PrevStatCodeConn
   IF "TRUE" THEN #"H_VDComMasterPNS7-1500".H_PrevStatCodeConn[1].H_Int := #TCON.Status_Mem; END_IF;
END_REGION

REGION Network 88: **** 8 - Outputs **** Return receive status code PrevStatCodeDisconn
   // Return receive status code H_PrevStatCodeDisconn
   IF "TRUE" THEN #"H_VDComMasterPNS7-1500".H_PrevStatCodeDisconn[1].H_Int := #TDISCON.Status_Mem; END_IF;
END_REGION

REGION Network 89: **** 8 - Outputs **** Return send status code PrevStatCodeRecv
   // Return send status code H_PrevStatCodeRecv
   IF "TRUE" THEN #"H_VDComMasterPNS7-1500".H_PrevStatCodeRecv[1].H_Int := #TRECV.Status_Mem; END_IF;
END_REGION

REGION Network 90: **** 8 - Outputs **** Return send status code PrevStatCodeSend
   // Return send status code H_PrevStatCodeSend
   IF "TRUE" THEN #"H_VDComMasterPNS7-1500".H_PrevStatCodeSend[1].H_Int := #TSEND.Status_Mem; END_IF;
END_REGION

REGION Network 91: **** 8 - Outputs **** New Message
   // New Message
   #IO_VD.NewMessageVD := #NewMessage;
END_REGION

REGION Network 92: **** 9 - Alarm Summary **** Alarm A
   // Alarm A
   #AlarmA := "FALSE";
END_REGION

REGION Network 93: **** 9 - Alarm Summary **** Alarm B
   // Alarm B
   #AlarmB := "FALSE";
END_REGION

REGION Network 94: **** 9 - Alarm Summary **** Alarm C
   // Alarm C
   #AlarmC := "FALSE";
END_REGION

REGION Network 95: **** 9 - Alarm Summary **** Alarm D
   // Alarm D
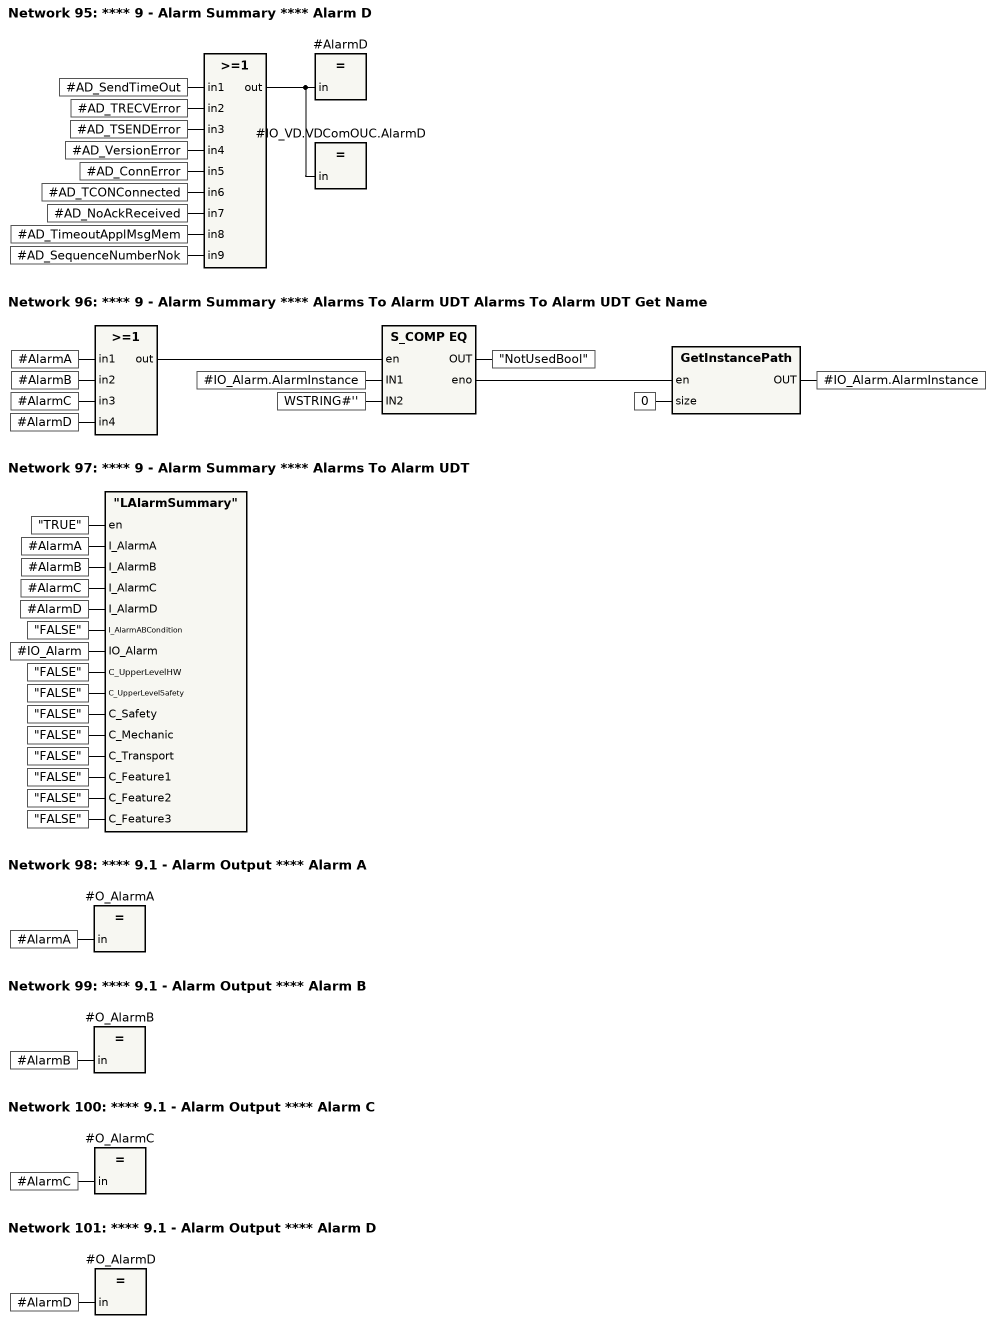
   #AlarmD := #AD_SendTimeOut OR #AD_TRECVError OR #AD_TSENDError OR #AD_VersionError OR #AD_ConnError OR #AD_TCONConnected OR #AD_NoAckReceived OR #AD_TimeoutApplMsgMem OR #AD_SequenceNumberNok;
   #IO_VD.VDComOUC.AlarmD := #AlarmD;
END_REGION

REGION Network 96: **** 9 - Alarm Summary **** Alarms To Alarm UDT Alarms To Alarm UDT Get Name
   // Alarm / Alarm D
   S_COMP(EN := #AlarmA OR #AlarmB OR #AlarmC OR #AlarmD,
          IN1 := #IO_Alarm.AlarmInstance,
          IN2 := WSTRING#'',
          OUT => "NotUsedBool",
          ENO => #_w1);
   IF #_w1 THEN GetInstancePath(size := 0, OUT => #IO_Alarm.AlarmInstance); END_IF;
END_REGION

REGION Network 97: **** 9 - Alarm Summary **** Alarms To Alarm UDT
   // Alarm / Alarm D
   IF "TRUE" THEN
       "LAlarmSummary"(I_AlarmA := #AlarmA,
                       I_AlarmB := #AlarmB,
                       I_AlarmC := #AlarmC,
                       I_AlarmD := #AlarmD,
                       I_AlarmABCondition := "FALSE",
                       IO_Alarm := #IO_Alarm,
                       C_UpperLevelHW := "FALSE",
                       C_UpperLevelSafety := "FALSE",
                       C_Safety := "FALSE",
                       C_Mechanic := "FALSE",
                       C_Transport := "FALSE",
                       C_Feature1 := "FALSE",
                       C_Feature2 := "FALSE",
                       C_Feature3 := "FALSE");
   END_IF;
END_REGION

REGION Network 98: **** 9.1 - Alarm Output **** Alarm A
   // Alarm A
   #O_AlarmA := #AlarmA;
END_REGION

REGION Network 99: **** 9.1 - Alarm Output **** Alarm B
   // Alarm B
   #O_AlarmB := #AlarmB;
END_REGION

REGION Network 100: **** 9.1 - Alarm Output **** Alarm C
   // Alarm C
   #O_AlarmC := #AlarmC;
END_REGION

REGION Network 101: **** 9.1 - Alarm Output **** Alarm D
   // Alarm D
   #O_AlarmD := #AlarmD;
END_REGION

REGION Network 102: **** 9.2 - Alarm DWord**** Alarm To DWord
   // Alarm To Word
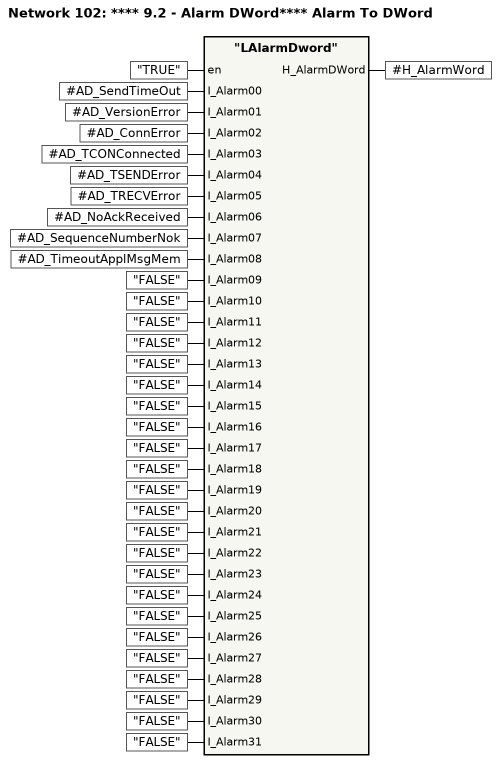
   IF "TRUE" THEN
       "LAlarmDword"(I_Alarm00 := #AD_SendTimeOut,
                     I_Alarm01 := #AD_VersionError,
                     I_Alarm02 := #AD_ConnError,
                     I_Alarm03 := #AD_TCONConnected,
                     I_Alarm04 := #AD_TSENDError,
                     I_Alarm05 := #AD_TRECVError,
                     I_Alarm06 := #AD_NoAckReceived,
                     I_Alarm07 := #AD_SequenceNumberNok,
                     I_Alarm08 := #AD_TimeoutApplMsgMem,
                     I_Alarm09 := "FALSE",
                     I_Alarm10 := "FALSE",
                     I_Alarm11 := "FALSE",
                     I_Alarm12 := "FALSE",
                     I_Alarm13 := "FALSE",
                     I_Alarm14 := "FALSE",
                     I_Alarm15 := "FALSE",
                     I_Alarm16 := "FALSE",
                     I_Alarm17 := "FALSE",
                     I_Alarm18 := "FALSE",
                     I_Alarm19 := "FALSE",
                     I_Alarm20 := "FALSE",
                     I_Alarm21 := "FALSE",
                     I_Alarm22 := "FALSE",
                     I_Alarm23 := "FALSE",
                     I_Alarm24 := "FALSE",
                     I_Alarm25 := "FALSE",
                     I_Alarm26 := "FALSE",
                     I_Alarm27 := "FALSE",
                     I_Alarm28 := "FALSE",
                     I_Alarm29 := "FALSE",
                     I_Alarm30 := "FALSE",
                     I_Alarm31 := "FALSE",
                     H_AlarmDWord => #H_AlarmWord);
   END_IF;
END_REGION
END_FUNCTION_BLOCK
